ABB RAPID module: StraightAlign3DP.modx

MODULE StraightAlign3DP


	VAR jointtarget CDP_0 := [[-10.64, 35.57, 6.66, 0, 47.77, -100.64], [9E9, 9E9, 9E9, 9E9, 9E9, 9E9]];
	VAR jointtarget CDP_1 := [[-9.53, 35.36, 7.02, 0, 47.62, -99.53], [9E9, 9E9, 9E9, 9E9, 9E9, 9E9]];
	VAR jointtarget CDP_2 := [[-8.41, 35.18, 7.34, 0, 47.48, -98.41], [9E9, 9E9, 9E9, 9E9, 9E9, 9E9]];
	VAR jointtarget CDP_3 := [[-7.29, 35.01, 7.62, 0, 47.37, -97.29], [9E9, 9E9, 9E9, 9E9, 9E9, 9E9]];
	VAR jointtarget CDP_4 := [[-6.16, 34.87, 7.86, 0, 47.27, -96.16], [9E9, 9E9, 9E9, 9E9, 9E9, 9E9]];
	VAR jointtarget CDP_5 := [[-5.02, 34.75, 8.06, 0, 47.19, -95.02], [9E9, 9E9, 9E9, 9E9, 9E9, 9E9]];
	VAR jointtarget CDP_6 := [[-3.89, 34.66, 8.22, 0, 47.12, -93.89], [9E9, 9E9, 9E9, 9E9, 9E9, 9E9]];
	VAR jointtarget CDP_7 := [[-2.75, 34.59, 8.33, 0, 47.07, -92.75], [9E9, 9E9, 9E9, 9E9, 9E9, 9E9]];
	VAR jointtarget CDP_8 := [[-1.6, 34.55, 8.41, 0, 47.04, -91.6], [9E9, 9E9, 9E9, 9E9, 9E9, 9E9]];
	VAR jointtarget CDP_9 := [[-0.46, 34.53, 8.45, 0, 47.03, -90.46], [9E9, 9E9, 9E9, 9E9, 9E9, 9E9]];
	VAR jointtarget CDP_10 := [[0.69, 34.53, 8.44, 0, 47.03, -89.31], [9E9, 9E9, 9E9, 9E9, 9E9, 9E9]];
	VAR jointtarget CDP_11 := [[1.83, 34.55, 8.4, 0, 47.05, -88.17], [9E9, 9E9, 9E9, 9E9, 9E9, 9E9]];
	VAR jointtarget CDP_12 := [[2.97, 34.6, 8.31, 0, 47.08, -87.03], [9E9, 9E9, 9E9, 9E9, 9E9, 9E9]];
	VAR jointtarget CDP_13 := [[4.11, 34.68, 8.19, 0, 47.13, -85.89], [9E9, 9E9, 9E9, 9E9, 9E9, 9E9]];
	VAR jointtarget CDP_14 := [[5.25, 34.78, 8.02, 0, 47.2, -84.75], [9E9, 9E9, 9E9, 9E9, 9E9, 9E9]];
	VAR jointtarget CDP_15 := [[6.38, 34.9, 7.82, 0, 47.29, -83.62], [9E9, 9E9, 9E9, 9E9, 9E9, 9E9]];
	VAR jointtarget CDP_16 := [[7.51, 35.04, 7.57, 0, 47.39, -82.49], [9E9, 9E9, 9E9, 9E9, 9E9, 9E9]];
	VAR jointtarget CDP_17 := [[8.63, 35.21, 7.28, 0, 47.51, -81.37], [9E9, 9E9, 9E9, 9E9, 9E9, 9E9]];
	VAR jointtarget CDP_18 := [[9.75, 35.4, 6.95, 0, 47.64, -80.25], [9E9, 9E9, 9E9, 9E9, 9E9, 9E9]];
	VAR jointtarget CDP_19 := [[10.86, 35.62, 6.58, 0, 47.8, -79.14], [9E9, 9E9, 9E9, 9E9, 9E9, 9E9]];
	VAR jointtarget CDP_20 := [[10.87, 35.62, 6.58, 0, 47.8, -79.46], [9E9, 9E9, 9E9, 9E9, 9E9, 9E9]];
	VAR jointtarget CDP_21 := [[10.89, 35.62, 6.57, 0, 47.8, -80.1], [9E9, 9E9, 9E9, 9E9, 9E9, 9E9]];
	VAR jointtarget CDP_22 := [[10.91, 35.63, 6.57, 0, 47.8, -80.75], [9E9, 9E9, 9E9, 9E9, 9E9, 9E9]];
	VAR jointtarget CDP_23 := [[10.92, 35.63, 6.56, 0, 47.81, -81.39], [9E9, 9E9, 9E9, 9E9, 9E9, 9E9]];
	VAR jointtarget CDP_24 := [[10.94, 35.63, 6.56, 0, 47.81, -82.04], [9E9, 9E9, 9E9, 9E9, 9E9, 9E9]];
	VAR jointtarget CDP_25 := [[10.96, 35.63, 6.56, 0, 47.81, -82.68], [9E9, 9E9, 9E9, 9E9, 9E9, 9E9]];
	VAR jointtarget CDP_26 := [[10.97, 35.64, 6.55, 0, 47.81, -83.33], [9E9, 9E9, 9E9, 9E9, 9E9, 9E9]];
	VAR jointtarget CDP_27 := [[10.99, 35.64, 6.55, 0, 47.81, -83.97], [9E9, 9E9, 9E9, 9E9, 9E9, 9E9]];
	VAR jointtarget CDP_28 := [[11.01, 35.64, 6.55, 0, 47.81, -84.62], [9E9, 9E9, 9E9, 9E9, 9E9, 9E9]];
	VAR jointtarget CDP_29 := [[11.02, 35.64, 6.54, 0, 47.81, -85.27], [9E9, 9E9, 9E9, 9E9, 9E9, 9E9]];
	VAR jointtarget CDP_30 := [[11.04, 35.64, 6.54, 0, 47.82, -85.91], [9E9, 9E9, 9E9, 9E9, 9E9, 9E9]];
	VAR jointtarget CDP_31 := [[11.06, 35.64, 6.54, 0, 47.82, -86.56], [9E9, 9E9, 9E9, 9E9, 9E9, 9E9]];
	VAR jointtarget CDP_32 := [[11.07, 35.65, 6.54, 0, 47.82, -87.2], [9E9, 9E9, 9E9, 9E9, 9E9, 9E9]];
	VAR jointtarget CDP_33 := [[11.09, 35.65, 6.54, 0, 47.82, -87.85], [9E9, 9E9, 9E9, 9E9, 9E9, 9E9]];
	VAR jointtarget CDP_34 := [[11.11, 35.65, 6.54, 0, 47.82, -88.49], [9E9, 9E9, 9E9, 9E9, 9E9, 9E9]];
	VAR jointtarget CDP_35 := [[11.13, 35.65, 6.54, 0, 47.82, -89.14], [9E9, 9E9, 9E9, 9E9, 9E9, 9E9]];
	VAR jointtarget CDP_36 := [[11.14, 35.65, 6.54, 0, 47.82, -89.78], [9E9, 9E9, 9E9, 9E9, 9E9, 9E9]];
	VAR jointtarget CDP_37 := [[11.16, 35.65, 6.54, 0, 47.82, -90.43], [9E9, 9E9, 9E9, 9E9, 9E9, 9E9]];
	VAR jointtarget CDP_38 := [[11.18, 35.65, 6.54, 0, 47.82, -91.07], [9E9, 9E9, 9E9, 9E9, 9E9, 9E9]];
	VAR jointtarget CDP_39 := [[11.19, 35.65, 6.54, 0, 47.82, -91.72], [9E9, 9E9, 9E9, 9E9, 9E9, 9E9]];
	VAR jointtarget CDP_40 := [[11.26, 35.64, 6.54, 0, 47.82, -91.98], [9E9, 9E9, 9E9, 9E9, 9E9, 9E9]];
	VAR jointtarget CDP_41 := [[11.33, 35.64, 6.55, 0, 47.81, -91.91], [9E9, 9E9, 9E9, 9E9, 9E9, 9E9]];
	VAR jointtarget CDP_42 := [[11.4, 35.64, 6.55, 0, 47.81, -91.84], [9E9, 9E9, 9E9, 9E9, 9E9, 9E9]];
	VAR jointtarget CDP_43 := [[11.47, 35.64, 6.55, 0, 47.81, -91.78], [9E9, 9E9, 9E9, 9E9, 9E9, 9E9]];
	VAR jointtarget CDP_44 := [[11.53, 35.63, 6.56, 0, 47.81, -91.71], [9E9, 9E9, 9E9, 9E9, 9E9, 9E9]];
	VAR jointtarget CDP_45 := [[11.6, 35.63, 6.56, 0, 47.81, -91.64], [9E9, 9E9, 9E9, 9E9, 9E9, 9E9]];
	VAR jointtarget CDP_46 := [[11.67, 35.63, 6.56, 0, 47.81, -91.57], [9E9, 9E9, 9E9, 9E9, 9E9, 9E9]];
	VAR jointtarget CDP_47 := [[11.74, 35.63, 6.57, 0, 47.8, -91.5], [9E9, 9E9, 9E9, 9E9, 9E9, 9E9]];
	VAR jointtarget CDP_48 := [[11.81, 35.63, 6.57, 0, 47.8, -91.44], [9E9, 9E9, 9E9, 9E9, 9E9, 9E9]];
	VAR jointtarget CDP_49 := [[11.87, 35.62, 6.57, 0, 47.8, -91.37], [9E9, 9E9, 9E9, 9E9, 9E9, 9E9]];
	VAR jointtarget CDP_50 := [[11.94, 35.62, 6.58, 0, 47.8, -91.3], [9E9, 9E9, 9E9, 9E9, 9E9, 9E9]];
	VAR jointtarget CDP_51 := [[12.01, 35.62, 6.58, 0, 47.8, -91.23], [9E9, 9E9, 9E9, 9E9, 9E9, 9E9]];
	VAR jointtarget CDP_52 := [[12.08, 35.62, 6.58, 0, 47.8, -91.16], [9E9, 9E9, 9E9, 9E9, 9E9, 9E9]];
	VAR jointtarget CDP_53 := [[12.15, 35.62, 6.58, 0, 47.8, -91.09], [9E9, 9E9, 9E9, 9E9, 9E9, 9E9]];
	VAR jointtarget CDP_54 := [[12.21, 35.62, 6.59, 0, 47.8, -91.03], [9E9, 9E9, 9E9, 9E9, 9E9, 9E9]];
	VAR jointtarget CDP_55 := [[12.28, 35.62, 6.59, 0, 47.8, -90.96], [9E9, 9E9, 9E9, 9E9, 9E9, 9E9]];
	VAR jointtarget CDP_56 := [[12.35, 35.61, 6.59, 0, 47.79, -90.89], [9E9, 9E9, 9E9, 9E9, 9E9, 9E9]];
	VAR jointtarget CDP_57 := [[12.42, 35.61, 6.59, 0, 47.79, -90.82], [9E9, 9E9, 9E9, 9E9, 9E9, 9E9]];
	VAR jointtarget CDP_58 := [[12.49, 35.61, 6.59, 0, 47.79, -90.75], [9E9, 9E9, 9E9, 9E9, 9E9, 9E9]];
	VAR jointtarget CDP_59 := [[12.55, 35.61, 6.6, 0, 47.79, -90.69], [9E9, 9E9, 9E9, 9E9, 9E9, 9E9]];
	VAR jointtarget CDP_60 := [[12.69, 35.62, 6.58, 0, 47.8, -85.39], [9E9, 9E9, 9E9, 9E9, 9E9, 9E9]];
	VAR jointtarget CDP_61 := [[12.81, 35.66, 6.51, 0, 47.83, -74.94], [9E9, 9E9, 9E9, 9E9, 9E9, 9E9]];
	VAR jointtarget CDP_62 := [[12.93, 35.72, 6.41, 0, 47.87, -64.5], [9E9, 9E9, 9E9, 9E9, 9E9, 9E9]];
	VAR jointtarget CDP_63 := [[13.04, 35.8, 6.27, 0, 47.93, -54.07], [9E9, 9E9, 9E9, 9E9, 9E9, 9E9]];
	VAR jointtarget CDP_64 := [[13.13, 35.91, 6.09, 0, 48, -43.65], [9E9, 9E9, 9E9, 9E9, 9E9, 9E9]];
	VAR jointtarget CDP_65 := [[13.2, 36.02, 5.89, 0, 48.09, -33.25], [9E9, 9E9, 9E9, 9E9, 9E9, 9E9]];
	VAR jointtarget CDP_66 := [[13.25, 36.16, 5.66, 0, 48.18, -22.88], [9E9, 9E9, 9E9, 9E9, 9E9, 9E9]];
	VAR jointtarget CDP_67 := [[13.28, 36.3, 5.42, 0, 48.28, -12.53], [9E9, 9E9, 9E9, 9E9, 9E9, 9E9]];
	VAR jointtarget CDP_68 := [[13.29, 36.44, 5.18, 0, 48.38, -2.2], [9E9, 9E9, 9E9, 9E9, 9E9, 9E9]];
	VAR jointtarget CDP_69 := [[13.27, 36.58, 4.93, 0, 48.49, 8.11], [9E9, 9E9, 9E9, 9E9, 9E9, 9E9]];
	VAR jointtarget CDP_70 := [[13.23, 36.71, 4.7, 0, 48.58, 18.39], [9E9, 9E9, 9E9, 9E9, 9E9, 9E9]];
	VAR jointtarget CDP_71 := [[13.17, 36.84, 4.48, 0, 48.68, 28.65], [9E9, 9E9, 9E9, 9E9, 9E9, 9E9]];
	VAR jointtarget CDP_72 := [[13.08, 36.95, 4.29, 0, 48.76, 38.9], [9E9, 9E9, 9E9, 9E9, 9E9, 9E9]];
	VAR jointtarget CDP_73 := [[12.99, 37.05, 4.13, 0, 48.82, 49.12], [9E9, 9E9, 9E9, 9E9, 9E9, 9E9]];
	VAR jointtarget CDP_74 := [[12.88, 37.12, 4, 0, 48.88, 59.33], [9E9, 9E9, 9E9, 9E9, 9E9, 9E9]];
	VAR jointtarget CDP_75 := [[12.75, 37.17, 3.92, 0, 48.91, 69.54], [9E9, 9E9, 9E9, 9E9, 9E9, 9E9]];
	VAR jointtarget CDP_76 := [[12.63, 37.19, 3.87, 0, 48.93, 79.73], [9E9, 9E9, 9E9, 9E9, 9E9, 9E9]];
	VAR jointtarget CDP_77 := [[12.5, 37.19, 3.87, 0, 48.93, 89.93], [9E9, 9E9, 9E9, 9E9, 9E9, 9E9]];
	VAR jointtarget CDP_78 := [[12.37, 37.17, 3.92, 0, 48.91, 100.13], [9E9, 9E9, 9E9, 9E9, 9E9, 9E9]];
	VAR jointtarget CDP_79 := [[12.25, 37.12, 4, 0, 48.88, 110.33], [9E9, 9E9, 9E9, 9E9, 9E9, 9E9]];
	VAR jointtarget CDP_80 := [[12.19, 37.09, 4.06, 0, 48.85, 115.43], [9E9, 9E9, 9E9, 9E9, 9E9, 9E9]];
	VAR jointtarget CDP_81 := [[12.13, 37.06, 4.11, 0, 48.83, 115.37], [9E9, 9E9, 9E9, 9E9, 9E9, 9E9]];
	VAR jointtarget CDP_82 := [[12.07, 37.02, 4.17, 0, 48.81, 115.31], [9E9, 9E9, 9E9, 9E9, 9E9, 9E9]];
	VAR jointtarget CDP_83 := [[12.01, 36.99, 4.22, 0, 48.79, 115.25], [9E9, 9E9, 9E9, 9E9, 9E9, 9E9]];
	VAR jointtarget CDP_84 := [[11.95, 36.96, 4.28, 0, 48.76, 115.19], [9E9, 9E9, 9E9, 9E9, 9E9, 9E9]];
	VAR jointtarget CDP_85 := [[11.89, 36.93, 4.33, 0, 48.74, 115.13], [9E9, 9E9, 9E9, 9E9, 9E9, 9E9]];
	VAR jointtarget CDP_86 := [[11.83, 36.9, 4.38, 0, 48.72, 115.07], [9E9, 9E9, 9E9, 9E9, 9E9, 9E9]];
	VAR jointtarget CDP_87 := [[11.77, 36.87, 4.44, 0, 48.7, 115.01], [9E9, 9E9, 9E9, 9E9, 9E9, 9E9]];
	VAR jointtarget CDP_88 := [[11.71, 36.84, 4.49, 0, 48.67, 114.95], [9E9, 9E9, 9E9, 9E9, 9E9, 9E9]];
	VAR jointtarget CDP_89 := [[11.65, 36.81, 4.54, 0, 48.65, 114.89], [9E9, 9E9, 9E9, 9E9, 9E9, 9E9]];
	VAR jointtarget CDP_90 := [[11.59, 36.77, 4.6, 0, 48.63, 114.83], [9E9, 9E9, 9E9, 9E9, 9E9, 9E9]];
	VAR jointtarget CDP_91 := [[11.53, 36.74, 4.65, 0, 48.61, 114.77], [9E9, 9E9, 9E9, 9E9, 9E9, 9E9]];
	VAR jointtarget CDP_92 := [[11.47, 36.71, 4.7, 0, 48.58, 114.71], [9E9, 9E9, 9E9, 9E9, 9E9, 9E9]];
	VAR jointtarget CDP_93 := [[11.4, 36.68, 4.76, 0, 48.56, 114.64], [9E9, 9E9, 9E9, 9E9, 9E9, 9E9]];
	VAR jointtarget CDP_94 := [[11.34, 36.65, 4.81, 0, 48.54, 114.58], [9E9, 9E9, 9E9, 9E9, 9E9, 9E9]];
	VAR jointtarget CDP_95 := [[11.28, 36.62, 4.86, 0, 48.52, 114.52], [9E9, 9E9, 9E9, 9E9, 9E9, 9E9]];
	VAR jointtarget CDP_96 := [[11.22, 36.59, 4.92, 0, 48.49, 114.46], [9E9, 9E9, 9E9, 9E9, 9E9, 9E9]];
	VAR jointtarget CDP_97 := [[11.16, 36.56, 4.97, 0, 48.47, 114.4], [9E9, 9E9, 9E9, 9E9, 9E9, 9E9]];
	VAR jointtarget CDP_98 := [[11.1, 36.53, 5.02, 0, 48.45, 114.34], [9E9, 9E9, 9E9, 9E9, 9E9, 9E9]];
	VAR jointtarget CDP_99 := [[11.04, 36.5, 5.07, 0, 48.43, 114.28], [9E9, 9E9, 9E9, 9E9, 9E9, 9E9]];
	VAR jointtarget CDP_100 := [[11.02, 36.49, 5.08, 0, 48.42, 113.93], [9E9, 9E9, 9E9, 9E9, 9E9, 9E9]];
	VAR jointtarget CDP_101 := [[11.01, 36.48, 5.1, 0, 48.42, 113.26], [9E9, 9E9, 9E9, 9E9, 9E9, 9E9]];
	VAR jointtarget CDP_102 := [[10.99, 36.48, 5.11, 0, 48.41, 112.58], [9E9, 9E9, 9E9, 9E9, 9E9, 9E9]];
	VAR jointtarget CDP_103 := [[10.98, 36.47, 5.12, 0, 48.41, 111.9], [9E9, 9E9, 9E9, 9E9, 9E9, 9E9]];
	VAR jointtarget CDP_104 := [[10.96, 36.46, 5.13, 0, 48.4, 111.22], [9E9, 9E9, 9E9, 9E9, 9E9, 9E9]];
	VAR jointtarget CDP_105 := [[10.95, 36.46, 5.14, 0, 48.4, 110.55], [9E9, 9E9, 9E9, 9E9, 9E9, 9E9]];
	VAR jointtarget CDP_106 := [[10.93, 36.45, 5.15, 0, 48.39, 109.87], [9E9, 9E9, 9E9, 9E9, 9E9, 9E9]];
	VAR jointtarget CDP_107 := [[10.91, 36.45, 5.16, 0, 48.39, 109.19], [9E9, 9E9, 9E9, 9E9, 9E9, 9E9]];
	VAR jointtarget CDP_108 := [[10.9, 36.44, 5.17, 0, 48.39, 108.51], [9E9, 9E9, 9E9, 9E9, 9E9, 9E9]];
	VAR jointtarget CDP_109 := [[10.88, 36.43, 5.18, 0, 48.38, 107.83], [9E9, 9E9, 9E9, 9E9, 9E9, 9E9]];
	VAR jointtarget CDP_110 := [[10.87, 36.43, 5.19, 0, 48.38, 107.16], [9E9, 9E9, 9E9, 9E9, 9E9, 9E9]];
	VAR jointtarget CDP_111 := [[10.85, 36.42, 5.2, 0, 48.37, 106.48], [9E9, 9E9, 9E9, 9E9, 9E9, 9E9]];
	VAR jointtarget CDP_112 := [[10.83, 36.42, 5.21, 0, 48.37, 105.8], [9E9, 9E9, 9E9, 9E9, 9E9, 9E9]];
	VAR jointtarget CDP_113 := [[10.82, 36.41, 5.22, 0, 48.37, 105.12], [9E9, 9E9, 9E9, 9E9, 9E9, 9E9]];
	VAR jointtarget CDP_114 := [[10.8, 36.41, 5.23, 0, 48.36, 104.44], [9E9, 9E9, 9E9, 9E9, 9E9, 9E9]];
	VAR jointtarget CDP_115 := [[10.79, 36.4, 5.23, 0, 48.36, 103.77], [9E9, 9E9, 9E9, 9E9, 9E9, 9E9]];
	VAR jointtarget CDP_116 := [[10.77, 36.4, 5.24, 0, 48.36, 103.09], [9E9, 9E9, 9E9, 9E9, 9E9, 9E9]];
	VAR jointtarget CDP_117 := [[10.75, 36.4, 5.25, 0, 48.36, 102.41], [9E9, 9E9, 9E9, 9E9, 9E9, 9E9]];
	VAR jointtarget CDP_118 := [[10.74, 36.39, 5.25, 0, 48.35, 101.73], [9E9, 9E9, 9E9, 9E9, 9E9, 9E9]];
	VAR jointtarget CDP_119 := [[10.72, 36.39, 5.26, 0, 48.35, 101.05], [9E9, 9E9, 9E9, 9E9, 9E9, 9E9]];
	VAR jointtarget CDP_120 := [[9.64, 36.18, 5.62, 0, 48.2, 99.64], [9E9, 9E9, 9E9, 9E9, 9E9, 9E9]];
	VAR jointtarget CDP_121 := [[8.56, 35.99, 5.95, 0, 48.06, 98.56], [9E9, 9E9, 9E9, 9E9, 9E9, 9E9]];
	VAR jointtarget CDP_122 := [[7.47, 35.83, 6.23, 0, 47.95, 97.47], [9E9, 9E9, 9E9, 9E9, 9E9, 9E9]];
	VAR jointtarget CDP_123 := [[6.38, 35.68, 6.47, 0, 47.84, 96.38], [9E9, 9E9, 9E9, 9E9, 9E9, 9E9]];
	VAR jointtarget CDP_124 := [[5.28, 35.56, 6.68, 0, 47.76, 95.28], [9E9, 9E9, 9E9, 9E9, 9E9, 9E9]];
	VAR jointtarget CDP_125 := [[4.17, 35.46, 6.85, 0, 47.69, 94.17], [9E9, 9E9, 9E9, 9E9, 9E9, 9E9]];
	VAR jointtarget CDP_126 := [[3.07, 35.39, 6.97, 0, 47.64, 93.07], [9E9, 9E9, 9E9, 9E9, 9E9, 9E9]];
	VAR jointtarget CDP_127 := [[1.96, 35.34, 7.06, 0, 47.6, 91.96], [9E9, 9E9, 9E9, 9E9, 9E9, 9E9]];
	VAR jointtarget CDP_128 := [[0.85, 35.31, 7.11, 0, 47.58, 90.85], [9E9, 9E9, 9E9, 9E9, 9E9, 9E9]];
	VAR jointtarget CDP_129 := [[-0.26, 35.3, 7.12, 0, 47.57, 89.74], [9E9, 9E9, 9E9, 9E9, 9E9, 9E9]];
	VAR jointtarget CDP_130 := [[-1.37, 35.32, 7.09, 0, 47.59, 88.63], [9E9, 9E9, 9E9, 9E9, 9E9, 9E9]];
	VAR jointtarget CDP_131 := [[-2.48, 35.36, 7.03, 0, 47.61, 87.52], [9E9, 9E9, 9E9, 9E9, 9E9, 9E9]];
	VAR jointtarget CDP_132 := [[-3.59, 35.42, 6.92, 0, 47.66, 86.41], [9E9, 9E9, 9E9, 9E9, 9E9, 9E9]];
	VAR jointtarget CDP_133 := [[-4.7, 35.51, 6.77, 0, 47.72, 85.3], [9E9, 9E9, 9E9, 9E9, 9E9, 9E9]];
	VAR jointtarget CDP_134 := [[-5.8, 35.62, 6.59, 0, 47.8, 84.2], [9E9, 9E9, 9E9, 9E9, 9E9, 9E9]];
	VAR jointtarget CDP_135 := [[-6.9, 35.75, 6.36, 0, 47.89, 83.1], [9E9, 9E9, 9E9, 9E9, 9E9, 9E9]];
	VAR jointtarget CDP_136 := [[-7.99, 35.9, 6.1, 0, 48, 82.01], [9E9, 9E9, 9E9, 9E9, 9E9, 9E9]];
	VAR jointtarget CDP_137 := [[-9.08, 36.08, 5.8, 0, 48.13, 80.92], [9E9, 9E9, 9E9, 9E9, 9E9, 9E9]];
	VAR jointtarget CDP_138 := [[-10.16, 36.28, 5.46, 0, 48.27, 79.84], [9E9, 9E9, 9E9, 9E9, 9E9, 9E9]];
	VAR jointtarget CDP_139 := [[-11.23, 36.5, 5.07, 0, 48.43, 78.77], [9E9, 9E9, 9E9, 9E9, 9E9, 9E9]];
	VAR jointtarget CDP_140 := [[-11.28, 36.51, 5.06, 0, 48.44, 79.81], [9E9, 9E9, 9E9, 9E9, 9E9, 9E9]];
	VAR jointtarget CDP_141 := [[-11.34, 36.52, 5.04, 0, 48.44, 81.95], [9E9, 9E9, 9E9, 9E9, 9E9, 9E9]];
	VAR jointtarget CDP_142 := [[-11.39, 36.52, 5.03, 0, 48.45, 84.09], [9E9, 9E9, 9E9, 9E9, 9E9, 9E9]];
	VAR jointtarget CDP_143 := [[-11.45, 36.53, 5.02, 0, 48.45, 86.23], [9E9, 9E9, 9E9, 9E9, 9E9, 9E9]];
	VAR jointtarget CDP_144 := [[-11.5, 36.53, 5.02, 0, 48.45, 88.37], [9E9, 9E9, 9E9, 9E9, 9E9, 9E9]];
	VAR jointtarget CDP_145 := [[-11.56, 36.53, 5.02, 0, 48.45, 90.51], [9E9, 9E9, 9E9, 9E9, 9E9, 9E9]];
	VAR jointtarget CDP_146 := [[-11.61, 36.53, 5.03, 0, 48.45, 92.65], [9E9, 9E9, 9E9, 9E9, 9E9, 9E9]];
	VAR jointtarget CDP_147 := [[-11.67, 36.52, 5.04, 0, 48.44, 94.78], [9E9, 9E9, 9E9, 9E9, 9E9, 9E9]];
	VAR jointtarget CDP_148 := [[-11.72, 36.51, 5.05, 0, 48.44, 96.92], [9E9, 9E9, 9E9, 9E9, 9E9, 9E9]];
	VAR jointtarget CDP_149 := [[-11.78, 36.5, 5.06, 0, 48.43, 99.06], [9E9, 9E9, 9E9, 9E9, 9E9, 9E9]];
	VAR jointtarget CDP_150 := [[-11.83, 36.49, 5.09, 0, 48.42, 101.2], [9E9, 9E9, 9E9, 9E9, 9E9, 9E9]];
	VAR jointtarget CDP_151 := [[-11.89, 36.48, 5.11, 0, 48.41, 103.34], [9E9, 9E9, 9E9, 9E9, 9E9, 9E9]];
	VAR jointtarget CDP_152 := [[-11.94, 36.46, 5.14, 0, 48.4, 105.48], [9E9, 9E9, 9E9, 9E9, 9E9, 9E9]];
	VAR jointtarget CDP_153 := [[-11.99, 36.44, 5.17, 0, 48.39, 107.63], [9E9, 9E9, 9E9, 9E9, 9E9, 9E9]];
	VAR jointtarget CDP_154 := [[-12.04, 36.42, 5.2, 0, 48.37, 109.77], [9E9, 9E9, 9E9, 9E9, 9E9, 9E9]];
	VAR jointtarget CDP_155 := [[-12.09, 36.4, 5.24, 0, 48.36, 111.91], [9E9, 9E9, 9E9, 9E9, 9E9, 9E9]];
	VAR jointtarget CDP_156 := [[-12.15, 36.38, 5.28, 0, 48.34, 114.05], [9E9, 9E9, 9E9, 9E9, 9E9, 9E9]];
	VAR jointtarget CDP_157 := [[-12.19, 36.35, 5.33, 0, 48.32, 116.2], [9E9, 9E9, 9E9, 9E9, 9E9, 9E9]];
	VAR jointtarget CDP_158 := [[-12.24, 36.32, 5.38, 0, 48.3, 118.34], [9E9, 9E9, 9E9, 9E9, 9E9, 9E9]];
	VAR jointtarget CDP_159 := [[-12.29, 36.29, 5.43, 0, 48.28, 120.49], [9E9, 9E9, 9E9, 9E9, 9E9, 9E9]];
	VAR jointtarget CDP_160 := [[-12.32, 36.27, 5.47, 0, 48.26, 121.56], [9E9, 9E9, 9E9, 9E9, 9E9, 9E9]];
	VAR jointtarget CDP_161 := [[-12.35, 36.25, 5.5, 0, 48.25, 121.53], [9E9, 9E9, 9E9, 9E9, 9E9, 9E9]];
	VAR jointtarget CDP_162 := [[-12.38, 36.23, 5.53, 0, 48.24, 121.5], [9E9, 9E9, 9E9, 9E9, 9E9, 9E9]];
	VAR jointtarget CDP_163 := [[-12.41, 36.21, 5.56, 0, 48.22, 121.47], [9E9, 9E9, 9E9, 9E9, 9E9, 9E9]];
	VAR jointtarget CDP_164 := [[-12.43, 36.19, 5.6, 0, 48.21, 121.44], [9E9, 9E9, 9E9, 9E9, 9E9, 9E9]];
	VAR jointtarget CDP_165 := [[-12.46, 36.18, 5.63, 0, 48.2, 121.41], [9E9, 9E9, 9E9, 9E9, 9E9, 9E9]];
	VAR jointtarget CDP_166 := [[-12.49, 36.16, 5.66, 0, 48.18, 121.39], [9E9, 9E9, 9E9, 9E9, 9E9, 9E9]];
	VAR jointtarget CDP_167 := [[-12.52, 36.14, 5.69, 0, 48.17, 121.36], [9E9, 9E9, 9E9, 9E9, 9E9, 9E9]];
	VAR jointtarget CDP_168 := [[-12.55, 36.12, 5.73, 0, 48.16, 121.33], [9E9, 9E9, 9E9, 9E9, 9E9, 9E9]];
	VAR jointtarget CDP_169 := [[-12.58, 36.1, 5.76, 0, 48.14, 121.3], [9E9, 9E9, 9E9, 9E9, 9E9, 9E9]];
	VAR jointtarget CDP_170 := [[-12.61, 36.08, 5.79, 0, 48.13, 121.27], [9E9, 9E9, 9E9, 9E9, 9E9, 9E9]];
	VAR jointtarget CDP_171 := [[-12.63, 36.06, 5.82, 0, 48.11, 121.24], [9E9, 9E9, 9E9, 9E9, 9E9, 9E9]];
	VAR jointtarget CDP_172 := [[-12.66, 36.04, 5.86, 0, 48.1, 121.21], [9E9, 9E9, 9E9, 9E9, 9E9, 9E9]];
	VAR jointtarget CDP_173 := [[-12.69, 36.02, 5.89, 0, 48.09, 121.18], [9E9, 9E9, 9E9, 9E9, 9E9, 9E9]];
	VAR jointtarget CDP_174 := [[-12.72, 36.01, 5.92, 0, 48.07, 121.16], [9E9, 9E9, 9E9, 9E9, 9E9, 9E9]];
	VAR jointtarget CDP_175 := [[-12.75, 35.99, 5.95, 0, 48.06, 121.13], [9E9, 9E9, 9E9, 9E9, 9E9, 9E9]];
	VAR jointtarget CDP_176 := [[-12.78, 35.97, 5.99, 0, 48.05, 121.1], [9E9, 9E9, 9E9, 9E9, 9E9, 9E9]];
	VAR jointtarget CDP_177 := [[-12.81, 35.95, 6.02, 0, 48.03, 121.07], [9E9, 9E9, 9E9, 9E9, 9E9, 9E9]];
	VAR jointtarget CDP_178 := [[-12.84, 35.93, 6.05, 0, 48.02, 121.04], [9E9, 9E9, 9E9, 9E9, 9E9, 9E9]];
	VAR jointtarget CDP_179 := [[-12.86, 35.91, 6.08, 0, 48.01, 121.01], [9E9, 9E9, 9E9, 9E9, 9E9, 9E9]];
	VAR jointtarget CDP_180 := [[-13.02, 35.84, 6.21, 0, 47.95, 114.17], [9E9, 9E9, 9E9, 9E9, 9E9, 9E9]];
	VAR jointtarget CDP_181 := [[-13.18, 35.81, 6.26, 0, 47.93, 100.62], [9E9, 9E9, 9E9, 9E9, 9E9, 9E9]];
	VAR jointtarget CDP_182 := [[-13.34, 35.81, 6.25, 0, 47.94, 87.07], [9E9, 9E9, 9E9, 9E9, 9E9, 9E9]];
	VAR jointtarget CDP_183 := [[-13.5, 35.86, 6.16, 0, 47.97, 73.52], [9E9, 9E9, 9E9, 9E9, 9E9, 9E9]];
	VAR jointtarget CDP_184 := [[-13.64, 35.95, 6.01, 0, 48.04, 59.99], [9E9, 9E9, 9E9, 9E9, 9E9, 9E9]];
	VAR jointtarget CDP_185 := [[-13.76, 36.08, 5.8, 0, 48.12, 46.48], [9E9, 9E9, 9E9, 9E9, 9E9, 9E9]];
	VAR jointtarget CDP_186 := [[-13.85, 36.22, 5.54, 0, 48.23, 33.01], [9E9, 9E9, 9E9, 9E9, 9E9, 9E9]];
	VAR jointtarget CDP_187 := [[-13.91, 36.39, 5.26, 0, 48.35, 19.56], [9E9, 9E9, 9E9, 9E9, 9E9, 9E9]];
	VAR jointtarget CDP_188 := [[-13.92, 36.57, 4.95, 0, 48.48, 6.16], [9E9, 9E9, 9E9, 9E9, 9E9, 9E9]];
	VAR jointtarget CDP_189 := [[-13.9, 36.75, 4.64, 0, 48.61, -7.21], [9E9, 9E9, 9E9, 9E9, 9E9, 9E9]];
	VAR jointtarget CDP_190 := [[-13.85, 36.92, 4.36, 0, 48.73, -20.54], [9E9, 9E9, 9E9, 9E9, 9E9, 9E9]];
	VAR jointtarget CDP_191 := [[-13.76, 37.06, 4.1, 0, 48.84, -33.84], [9E9, 9E9, 9E9, 9E9, 9E9, 9E9]];
	VAR jointtarget CDP_192 := [[-13.64, 37.19, 3.89, 0, 48.93, -47.11], [9E9, 9E9, 9E9, 9E9, 9E9, 9E9]];
	VAR jointtarget CDP_193 := [[-13.5, 37.27, 3.73, 0, 48.99, -60.35], [9E9, 9E9, 9E9, 9E9, 9E9, 9E9]];
	VAR jointtarget CDP_194 := [[-13.34, 37.33, 3.65, 0, 49.03, -73.59], [9E9, 9E9, 9E9, 9E9, 9E9, 9E9]];
	VAR jointtarget CDP_195 := [[-13.18, 37.34, 3.63, 0, 49.04, -86.81], [9E9, 9E9, 9E9, 9E9, 9E9, 9E9]];
	VAR jointtarget CDP_196 := [[-13.02, 37.3, 3.68, 0, 49.01, -100.04], [9E9, 9E9, 9E9, 9E9, 9E9, 9E9]];
	VAR jointtarget CDP_197 := [[-12.88, 37.23, 3.81, 0, 48.96, -113.28], [9E9, 9E9, 9E9, 9E9, 9E9, 9E9]];
	VAR jointtarget CDP_198 := [[-12.75, 37.13, 3.99, 0, 48.88, -126.54], [9E9, 9E9, 9E9, 9E9, 9E9, 9E9]];
	VAR jointtarget CDP_199 := [[-12.64, 36.99, 4.23, 0, 48.78, -139.82], [9E9, 9E9, 9E9, 9E9, 9E9, 9E9]];
	VAR jointtarget CDP_200 := [[-12.62, 36.95, 4.3, 0, 48.75, -146.49], [9E9, 9E9, 9E9, 9E9, 9E9, 9E9]];
	VAR jointtarget CDP_201 := [[-12.59, 36.91, 4.37, 0, 48.72, -146.47], [9E9, 9E9, 9E9, 9E9, 9E9, 9E9]];
	VAR jointtarget CDP_202 := [[-12.57, 36.86, 4.44, 0, 48.69, -146.44], [9E9, 9E9, 9E9, 9E9, 9E9, 9E9]];
	VAR jointtarget CDP_203 := [[-12.54, 36.82, 4.51, 0, 48.66, -146.42], [9E9, 9E9, 9E9, 9E9, 9E9, 9E9]];
	VAR jointtarget CDP_204 := [[-12.52, 36.78, 4.58, 0, 48.63, -146.4], [9E9, 9E9, 9E9, 9E9, 9E9, 9E9]];
	VAR jointtarget CDP_205 := [[-12.49, 36.74, 4.65, 0, 48.6, -146.37], [9E9, 9E9, 9E9, 9E9, 9E9, 9E9]];
	VAR jointtarget CDP_206 := [[-12.47, 36.7, 4.73, 0, 48.57, -146.35], [9E9, 9E9, 9E9, 9E9, 9E9, 9E9]];
	VAR jointtarget CDP_207 := [[-12.44, 36.66, 4.8, 0, 48.54, -146.32], [9E9, 9E9, 9E9, 9E9, 9E9, 9E9]];
	VAR jointtarget CDP_208 := [[-12.42, 36.62, 4.87, 0, 48.52, -146.3], [9E9, 9E9, 9E9, 9E9, 9E9, 9E9]];
	VAR jointtarget CDP_209 := [[-12.39, 36.58, 4.94, 0, 48.49, -146.27], [9E9, 9E9, 9E9, 9E9, 9E9, 9E9]];
	VAR jointtarget CDP_210 := [[-12.37, 36.54, 5.01, 0, 48.46, -146.25], [9E9, 9E9, 9E9, 9E9, 9E9, 9E9]];
	VAR jointtarget CDP_211 := [[-12.34, 36.5, 5.08, 0, 48.43, -146.22], [9E9, 9E9, 9E9, 9E9, 9E9, 9E9]];
	VAR jointtarget CDP_212 := [[-12.32, 36.45, 5.15, 0, 48.4, -146.2], [9E9, 9E9, 9E9, 9E9, 9E9, 9E9]];
	VAR jointtarget CDP_213 := [[-12.29, 36.41, 5.22, 0, 48.37, -146.17], [9E9, 9E9, 9E9, 9E9, 9E9, 9E9]];
	VAR jointtarget CDP_214 := [[-12.27, 36.37, 5.29, 0, 48.34, -146.15], [9E9, 9E9, 9E9, 9E9, 9E9, 9E9]];
	VAR jointtarget CDP_215 := [[-12.24, 36.33, 5.36, 0, 48.31, -146.12], [9E9, 9E9, 9E9, 9E9, 9E9, 9E9]];
	VAR jointtarget CDP_216 := [[-12.22, 36.29, 5.43, 0, 48.28, -146.1], [9E9, 9E9, 9E9, 9E9, 9E9, 9E9]];
	VAR jointtarget CDP_217 := [[-12.19, 36.25, 5.5, 0, 48.25, -146.07], [9E9, 9E9, 9E9, 9E9, 9E9, 9E9]];
	VAR jointtarget CDP_218 := [[-12.17, 36.21, 5.57, 0, 48.22, -146.05], [9E9, 9E9, 9E9, 9E9, 9E9, 9E9]];
	VAR jointtarget CDP_219 := [[-12.14, 36.17, 5.64, 0, 48.19, -146.02], [9E9, 9E9, 9E9, 9E9, 9E9, 9E9]];
	VAR jointtarget CDP_220 := [[-12.14, 36.16, 5.66, 0, 48.18, -145.46], [9E9, 9E9, 9E9, 9E9, 9E9, 9E9]];
	VAR jointtarget CDP_221 := [[-12.13, 36.14, 5.68, 0, 48.17, -144.35], [9E9, 9E9, 9E9, 9E9, 9E9, 9E9]];
	VAR jointtarget CDP_222 := [[-12.12, 36.13, 5.7, 0, 48.17, -143.24], [9E9, 9E9, 9E9, 9E9, 9E9, 9E9]];
	VAR jointtarget CDP_223 := [[-12.11, 36.12, 5.72, 0, 48.16, -142.13], [9E9, 9E9, 9E9, 9E9, 9E9, 9E9]];
	VAR jointtarget CDP_224 := [[-12.1, 36.11, 5.74, 0, 48.15, -141.01], [9E9, 9E9, 9E9, 9E9, 9E9, 9E9]];
	VAR jointtarget CDP_225 := [[-12.09, 36.1, 5.76, 0, 48.14, -139.9], [9E9, 9E9, 9E9, 9E9, 9E9, 9E9]];
	VAR jointtarget CDP_226 := [[-12.08, 36.08, 5.78, 0, 48.13, -138.79], [9E9, 9E9, 9E9, 9E9, 9E9, 9E9]];
	VAR jointtarget CDP_227 := [[-12.07, 36.07, 5.8, 0, 48.12, -137.68], [9E9, 9E9, 9E9, 9E9, 9E9, 9E9]];
	VAR jointtarget CDP_228 := [[-12.06, 36.06, 5.82, 0, 48.12, -136.56], [9E9, 9E9, 9E9, 9E9, 9E9, 9E9]];
	VAR jointtarget CDP_229 := [[-12.05, 36.05, 5.84, 0, 48.11, -135.45], [9E9, 9E9, 9E9, 9E9, 9E9, 9E9]];
	VAR jointtarget CDP_230 := [[-12.04, 36.04, 5.86, 0, 48.1, -134.34], [9E9, 9E9, 9E9, 9E9, 9E9, 9E9]];
	VAR jointtarget CDP_231 := [[-12.03, 36.03, 5.88, 0, 48.09, -133.22], [9E9, 9E9, 9E9, 9E9, 9E9, 9E9]];
	VAR jointtarget CDP_232 := [[-12.02, 36.02, 5.89, 0, 48.09, -132.11], [9E9, 9E9, 9E9, 9E9, 9E9, 9E9]];
	VAR jointtarget CDP_233 := [[-12.01, 36.01, 5.91, 0, 48.08, -130.99], [9E9, 9E9, 9E9, 9E9, 9E9, 9E9]];
	VAR jointtarget CDP_234 := [[-12, 36, 5.93, 0, 48.07, -129.88], [9E9, 9E9, 9E9, 9E9, 9E9, 9E9]];
	VAR jointtarget CDP_235 := [[-11.99, 35.99, 5.94, 0, 48.07, -128.76], [9E9, 9E9, 9E9, 9E9, 9E9, 9E9]];
	VAR jointtarget CDP_236 := [[-11.98, 35.98, 5.96, 0, 48.06, -127.65], [9E9, 9E9, 9E9, 9E9, 9E9, 9E9]];
	VAR jointtarget CDP_237 := [[-11.97, 35.97, 5.97, 0, 48.06, -126.53], [9E9, 9E9, 9E9, 9E9, 9E9, 9E9]];
	VAR jointtarget CDP_238 := [[-11.96, 35.96, 5.99, 0, 48.05, -125.42], [9E9, 9E9, 9E9, 9E9, 9E9, 9E9]];
	VAR jointtarget CDP_239 := [[-11.95, 35.95, 6, 0, 48.04, -124.3], [9E9, 9E9, 9E9, 9E9, 9E9, 9E9]];
	VAR jointtarget CDP_240 := [[-11.94, 35.94, 6.02, 0, 48.04, -123.74], [9E9, 9E9, 9E9, 9E9, 9E9, 9E9]];
	VAR jointtarget CDP_241 := [[-11.93, 35.94, 6.03, 0, 48.04, -123.73], [9E9, 9E9, 9E9, 9E9, 9E9, 9E9]];
	VAR jointtarget CDP_242 := [[-11.92, 35.93, 6.04, 0, 48.03, -123.72], [9E9, 9E9, 9E9, 9E9, 9E9, 9E9]];
	VAR jointtarget CDP_243 := [[-11.9, 35.92, 6.05, 0, 48.03, -123.71], [9E9, 9E9, 9E9, 9E9, 9E9, 9E9]];
	VAR jointtarget CDP_244 := [[-11.89, 35.91, 6.07, 0, 48.02, -123.7], [9E9, 9E9, 9E9, 9E9, 9E9, 9E9]];
	VAR jointtarget CDP_245 := [[-11.88, 35.9, 6.08, 0, 48.02, -123.69], [9E9, 9E9, 9E9, 9E9, 9E9, 9E9]];
	VAR jointtarget CDP_246 := [[-11.87, 35.9, 6.09, 0, 48.01, -123.68], [9E9, 9E9, 9E9, 9E9, 9E9, 9E9]];
	VAR jointtarget CDP_247 := [[-11.86, 35.89, 6.11, 0, 48.01, -123.66], [9E9, 9E9, 9E9, 9E9, 9E9, 9E9]];
	VAR jointtarget CDP_248 := [[-11.85, 35.88, 6.12, 0, 48, -123.65], [9E9, 9E9, 9E9, 9E9, 9E9, 9E9]];
	VAR jointtarget CDP_249 := [[-11.84, 35.87, 6.13, 0, 48, -123.64], [9E9, 9E9, 9E9, 9E9, 9E9, 9E9]];
	VAR jointtarget CDP_250 := [[-11.83, 35.86, 6.14, 0, 47.99, -123.63], [9E9, 9E9, 9E9, 9E9, 9E9, 9E9]];
	VAR jointtarget CDP_251 := [[-11.82, 35.86, 6.16, 0, 47.99, -123.62], [9E9, 9E9, 9E9, 9E9, 9E9, 9E9]];
	VAR jointtarget CDP_252 := [[-11.81, 35.85, 6.17, 0, 47.98, -123.61], [9E9, 9E9, 9E9, 9E9, 9E9, 9E9]];
	VAR jointtarget CDP_253 := [[-11.8, 35.84, 6.18, 0, 47.98, -123.6], [9E9, 9E9, 9E9, 9E9, 9E9, 9E9]];
	VAR jointtarget CDP_254 := [[-11.79, 35.83, 6.19, 0, 47.97, -123.59], [9E9, 9E9, 9E9, 9E9, 9E9, 9E9]];
	VAR jointtarget CDP_255 := [[-11.78, 35.83, 6.21, 0, 47.97, -123.58], [9E9, 9E9, 9E9, 9E9, 9E9, 9E9]];
	VAR jointtarget CDP_256 := [[-11.77, 35.82, 6.22, 0, 47.96, -123.57], [9E9, 9E9, 9E9, 9E9, 9E9, 9E9]];
	VAR jointtarget CDP_257 := [[-11.76, 35.81, 6.23, 0, 47.96, -123.56], [9E9, 9E9, 9E9, 9E9, 9E9, 9E9]];
	VAR jointtarget CDP_258 := [[-11.75, 35.8, 6.25, 0, 47.95, -123.55], [9E9, 9E9, 9E9, 9E9, 9E9, 9E9]];
	VAR jointtarget CDP_259 := [[-11.74, 35.79, 6.26, 0, 47.95, -123.54], [9E9, 9E9, 9E9, 9E9, 9E9, 9E9]];
	VAR jointtarget CDP_260 := [[-10.65, 35.56, 6.66, 0, 47.78, -100.65], [9E9, 9E9, 9E9, 9E9, 9E9, 9E9]];
	VAR jointtarget CDP_261 := [[-9.55, 35.35, 7.01, 0, 47.63, -99.55], [9E9, 9E9, 9E9, 9E9, 9E9, 9E9]];
	VAR jointtarget CDP_262 := [[-8.44, 35.17, 7.33, 0, 47.5, -98.44], [9E9, 9E9, 9E9, 9E9, 9E9, 9E9]];
	VAR jointtarget CDP_263 := [[-7.33, 35, 7.61, 0, 47.39, -97.33], [9E9, 9E9, 9E9, 9E9, 9E9, 9E9]];
	VAR jointtarget CDP_264 := [[-6.21, 34.86, 7.85, 0, 47.29, -96.21], [9E9, 9E9, 9E9, 9E9, 9E9, 9E9]];
	VAR jointtarget CDP_265 := [[-5.09, 34.75, 8.05, 0, 47.21, -95.09], [9E9, 9E9, 9E9, 9E9, 9E9, 9E9]];
	VAR jointtarget CDP_266 := [[-3.96, 34.65, 8.21, 0, 47.14, -93.96], [9E9, 9E9, 9E9, 9E9, 9E9, 9E9]];
	VAR jointtarget CDP_267 := [[-2.83, 34.58, 8.33, 0, 47.09, -92.83], [9E9, 9E9, 9E9, 9E9, 9E9, 9E9]];
	VAR jointtarget CDP_268 := [[-1.7, 34.54, 8.4, 0, 47.06, -91.7], [9E9, 9E9, 9E9, 9E9, 9E9, 9E9]];
	VAR jointtarget CDP_269 := [[-0.56, 34.51, 8.44, 0, 47.04, -90.56], [9E9, 9E9, 9E9, 9E9, 9E9, 9E9]];
	VAR jointtarget CDP_270 := [[0.57, 34.51, 8.44, 0, 47.04, -89.43], [9E9, 9E9, 9E9, 9E9, 9E9, 9E9]];
	VAR jointtarget CDP_271 := [[1.7, 34.54, 8.4, 0, 47.06, -88.3], [9E9, 9E9, 9E9, 9E9, 9E9, 9E9]];
	VAR jointtarget CDP_272 := [[2.84, 34.58, 8.32, 0, 47.09, -87.16], [9E9, 9E9, 9E9, 9E9, 9E9, 9E9]];
	VAR jointtarget CDP_273 := [[3.97, 34.65, 8.2, 0, 47.14, -86.03], [9E9, 9E9, 9E9, 9E9, 9E9, 9E9]];
	VAR jointtarget CDP_274 := [[5.09, 34.75, 8.05, 0, 47.21, -84.91], [9E9, 9E9, 9E9, 9E9, 9E9, 9E9]];
	VAR jointtarget CDP_275 := [[6.22, 34.86, 7.85, 0, 47.29, -83.78], [9E9, 9E9, 9E9, 9E9, 9E9, 9E9]];
	VAR jointtarget CDP_276 := [[7.34, 35, 7.61, 0, 47.39, -82.66], [9E9, 9E9, 9E9, 9E9, 9E9, 9E9]];
	VAR jointtarget CDP_277 := [[8.45, 35.17, 7.33, 0, 47.5, -81.55], [9E9, 9E9, 9E9, 9E9, 9E9, 9E9]];
	VAR jointtarget CDP_278 := [[9.56, 35.35, 7.01, 0, 47.64, -80.44], [9E9, 9E9, 9E9, 9E9, 9E9, 9E9]];
	VAR jointtarget CDP_279 := [[10.65, 35.56, 6.65, 0, 47.78, -79.35], [9E9, 9E9, 9E9, 9E9, 9E9, 9E9]];
	VAR jointtarget CDP_280 := [[10.71, 35.58, 6.63, 0, 47.79, -78.19], [9E9, 9E9, 9E9, 9E9, 9E9, 9E9]];
	VAR jointtarget CDP_281 := [[10.76, 35.59, 6.61, 0, 47.8, -75.95], [9E9, 9E9, 9E9, 9E9, 9E9, 9E9]];
	VAR jointtarget CDP_282 := [[10.82, 35.61, 6.58, 0, 47.82, -73.7], [9E9, 9E9, 9E9, 9E9, 9E9, 9E9]];
	VAR jointtarget CDP_283 := [[10.87, 35.63, 6.55, 0, 47.83, -71.45], [9E9, 9E9, 9E9, 9E9, 9E9, 9E9]];
	VAR jointtarget CDP_284 := [[10.92, 35.65, 6.51, 0, 47.84, -69.2], [9E9, 9E9, 9E9, 9E9, 9E9, 9E9]];
	VAR jointtarget CDP_285 := [[10.97, 35.67, 6.47, 0, 47.86, -66.96], [9E9, 9E9, 9E9, 9E9, 9E9, 9E9]];
	VAR jointtarget CDP_286 := [[11.03, 35.7, 6.42, 0, 47.88, -64.72], [9E9, 9E9, 9E9, 9E9, 9E9, 9E9]];
	VAR jointtarget CDP_287 := [[11.07, 35.72, 6.38, 0, 47.9, -62.47], [9E9, 9E9, 9E9, 9E9, 9E9, 9E9]];
	VAR jointtarget CDP_288 := [[11.12, 35.75, 6.33, 0, 47.92, -60.23], [9E9, 9E9, 9E9, 9E9, 9E9, 9E9]];
	VAR jointtarget CDP_289 := [[11.17, 35.79, 6.27, 0, 47.94, -57.99], [9E9, 9E9, 9E9, 9E9, 9E9, 9E9]];
	VAR jointtarget CDP_290 := [[11.22, 35.82, 6.21, 0, 47.97, -55.75], [9E9, 9E9, 9E9, 9E9, 9E9, 9E9]];
	VAR jointtarget CDP_291 := [[11.26, 35.86, 6.15, 0, 47.99, -53.51], [9E9, 9E9, 9E9, 9E9, 9E9, 9E9]];
	VAR jointtarget CDP_292 := [[11.3, 35.89, 6.09, 0, 48.02, -51.27], [9E9, 9E9, 9E9, 9E9, 9E9, 9E9]];
	VAR jointtarget CDP_293 := [[11.35, 35.93, 6.02, 0, 48.05, -49.04], [9E9, 9E9, 9E9, 9E9, 9E9, 9E9]];
	VAR jointtarget CDP_294 := [[11.39, 35.97, 5.95, 0, 48.08, -46.8], [9E9, 9E9, 9E9, 9E9, 9E9, 9E9]];
	VAR jointtarget CDP_295 := [[11.43, 36.02, 5.88, 0, 48.11, -44.57], [9E9, 9E9, 9E9, 9E9, 9E9, 9E9]];
	VAR jointtarget CDP_296 := [[11.46, 36.06, 5.8, 0, 48.14, -42.34], [9E9, 9E9, 9E9, 9E9, 9E9, 9E9]];
	VAR jointtarget CDP_297 := [[11.5, 36.11, 5.72, 0, 48.17, -40.11], [9E9, 9E9, 9E9, 9E9, 9E9, 9E9]];
	VAR jointtarget CDP_298 := [[11.53, 36.15, 5.64, 0, 48.21, -37.88], [9E9, 9E9, 9E9, 9E9, 9E9, 9E9]];
	VAR jointtarget CDP_299 := [[11.57, 36.2, 5.56, 0, 48.24, -35.65], [9E9, 9E9, 9E9, 9E9, 9E9, 9E9]];
	VAR jointtarget CDP_300 := [[11.59, 36.23, 5.5, 0, 48.26, -34.54], [9E9, 9E9, 9E9, 9E9, 9E9, 9E9]];
	VAR jointtarget CDP_301 := [[11.6, 36.26, 5.45, 0, 48.28, -34.52], [9E9, 9E9, 9E9, 9E9, 9E9, 9E9]];
	VAR jointtarget CDP_302 := [[11.62, 36.29, 5.4, 0, 48.31, -34.5], [9E9, 9E9, 9E9, 9E9, 9E9, 9E9]];
	VAR jointtarget CDP_303 := [[11.64, 36.32, 5.35, 0, 48.33, -34.48], [9E9, 9E9, 9E9, 9E9, 9E9, 9E9]];
	VAR jointtarget CDP_304 := [[11.66, 36.35, 5.3, 0, 48.35, -34.46], [9E9, 9E9, 9E9, 9E9, 9E9, 9E9]];
	VAR jointtarget CDP_305 := [[11.68, 36.38, 5.25, 0, 48.37, -34.44], [9E9, 9E9, 9E9, 9E9, 9E9, 9E9]];
	VAR jointtarget CDP_306 := [[11.7, 36.41, 5.19, 0, 48.39, -34.42], [9E9, 9E9, 9E9, 9E9, 9E9, 9E9]];
	VAR jointtarget CDP_307 := [[11.72, 36.44, 5.14, 0, 48.41, -34.41], [9E9, 9E9, 9E9, 9E9, 9E9, 9E9]];
	VAR jointtarget CDP_308 := [[11.74, 36.47, 5.09, 0, 48.44, -34.39], [9E9, 9E9, 9E9, 9E9, 9E9, 9E9]];
	VAR jointtarget CDP_309 := [[11.76, 36.5, 5.04, 0, 48.46, -34.37], [9E9, 9E9, 9E9, 9E9, 9E9, 9E9]];
	VAR jointtarget CDP_310 := [[11.77, 36.53, 4.99, 0, 48.48, -34.35], [9E9, 9E9, 9E9, 9E9, 9E9, 9E9]];
	VAR jointtarget CDP_311 := [[11.79, 36.56, 4.93, 0, 48.5, -34.33], [9E9, 9E9, 9E9, 9E9, 9E9, 9E9]];
	VAR jointtarget CDP_312 := [[11.81, 36.59, 4.88, 0, 48.52, -34.31], [9E9, 9E9, 9E9, 9E9, 9E9, 9E9]];
	VAR jointtarget CDP_313 := [[11.83, 36.62, 4.83, 0, 48.54, -34.29], [9E9, 9E9, 9E9, 9E9, 9E9, 9E9]];
	VAR jointtarget CDP_314 := [[11.85, 36.66, 4.78, 0, 48.57, -34.27], [9E9, 9E9, 9E9, 9E9, 9E9, 9E9]];
	VAR jointtarget CDP_315 := [[11.87, 36.69, 4.73, 0, 48.59, -34.26], [9E9, 9E9, 9E9, 9E9, 9E9, 9E9]];
	VAR jointtarget CDP_316 := [[11.89, 36.72, 4.67, 0, 48.61, -34.24], [9E9, 9E9, 9E9, 9E9, 9E9, 9E9]];
	VAR jointtarget CDP_317 := [[11.91, 36.75, 4.62, 0, 48.63, -34.22], [9E9, 9E9, 9E9, 9E9, 9E9, 9E9]];
	VAR jointtarget CDP_318 := [[11.92, 36.78, 4.57, 0, 48.65, -34.2], [9E9, 9E9, 9E9, 9E9, 9E9, 9E9]];
	VAR jointtarget CDP_319 := [[11.94, 36.81, 4.52, 0, 48.68, -34.18], [9E9, 9E9, 9E9, 9E9, 9E9, 9E9]];
	VAR jointtarget CDP_320 := [[12.05, 36.94, 4.28, 0, 48.77, -40.77], [9E9, 9E9, 9E9, 9E9, 9E9, 9E9]];
	VAR jointtarget CDP_321 := [[12.18, 37.05, 4.1, 0, 48.85, -54.03], [9E9, 9E9, 9E9, 9E9, 9E9, 9E9]];
	VAR jointtarget CDP_322 := [[12.33, 37.12, 3.98, 0, 48.9, -67.26], [9E9, 9E9, 9E9, 9E9, 9E9, 9E9]];
	VAR jointtarget CDP_323 := [[12.49, 37.15, 3.93, 0, 48.92, -80.49], [9E9, 9E9, 9E9, 9E9, 9E9, 9E9]];
	VAR jointtarget CDP_324 := [[12.65, 37.13, 3.95, 0, 48.91, -93.72], [9E9, 9E9, 9E9, 9E9, 9E9, 9E9]];
	VAR jointtarget CDP_325 := [[12.8, 37.08, 4.04, 0, 48.88, -106.95], [9E9, 9E9, 9E9, 9E9, 9E9, 9E9]];
	VAR jointtarget CDP_326 := [[12.94, 36.99, 4.2, 0, 48.81, -120.2], [9E9, 9E9, 9E9, 9E9, 9E9, 9E9]];
	VAR jointtarget CDP_327 := [[13.06, 36.87, 4.41, 0, 48.72, -133.47], [9E9, 9E9, 9E9, 9E9, 9E9, 9E9]];
	VAR jointtarget CDP_328 := [[13.15, 36.72, 4.67, 0, 48.61, -146.77], [9E9, 9E9, 9E9, 9E9, 9E9, 9E9]];
	VAR jointtarget CDP_329 := [[13.2, 36.55, 4.96, 0, 48.49, -160.1], [9E9, 9E9, 9E9, 9E9, 9E9, 9E9]];
	VAR jointtarget CDP_330 := [[13.22, 36.37, 5.27, 0, 48.36, -173.47], [9E9, 9E9, 9E9, 9E9, 9E9, 9E9]];
	VAR jointtarget CDP_331 := [[13.2, 36.19, 5.57, 0, 48.24, -186.88], [9E9, 9E9, 9E9, 9E9, 9E9, 9E9]];
	VAR jointtarget CDP_332 := [[13.15, 36.03, 5.86, 0, 48.12, -200.32], [9E9, 9E9, 9E9, 9E9, 9E9, 9E9]];
	VAR jointtarget CDP_333 := [[13.06, 35.88, 6.11, 0, 48.01, -213.8], [9E9, 9E9, 9E9, 9E9, 9E9, 9E9]];
	VAR jointtarget CDP_334 := [[12.93, 35.76, 6.32, 0, 47.92, -227.31], [9E9, 9E9, 9E9, 9E9, 9E9, 9E9]];
	VAR jointtarget CDP_335 := [[12.79, 35.67, 6.47, 0, 47.86, -240.84], [9E9, 9E9, 9E9, 9E9, 9E9, 9E9]];
	VAR jointtarget CDP_336 := [[12.63, 35.62, 6.55, 0, 47.83, -254.39], [9E9, 9E9, 9E9, 9E9, 9E9, 9E9]];
	VAR jointtarget CDP_337 := [[12.47, 35.62, 6.56, 0, 47.82, -267.94], [9E9, 9E9, 9E9, 9E9, 9E9, 9E9]];
	VAR jointtarget CDP_338 := [[12.3, 35.65, 6.5, 0, 47.85, -281.49], [9E9, 9E9, 9E9, 9E9, 9E9, 9E9]];
	VAR jointtarget CDP_339 := [[12.15, 35.73, 6.37, 0, 47.9, -295.03], [9E9, 9E9, 9E9, 9E9, 9E9, 9E9]];
	VAR jointtarget CDP_340 := [[12.13, 35.75, 6.34, 0, 47.91, -301.75], [9E9, 9E9, 9E9, 9E9, 9E9, 9E9]];
	VAR jointtarget CDP_341 := [[12.1, 35.77, 6.31, 0, 47.93, -301.78], [9E9, 9E9, 9E9, 9E9, 9E9, 9E9]];
	VAR jointtarget CDP_342 := [[12.07, 35.79, 6.27, 0, 47.94, -301.81], [9E9, 9E9, 9E9, 9E9, 9E9, 9E9]];
	VAR jointtarget CDP_343 := [[12.04, 35.8, 6.24, 0, 47.96, -301.84], [9E9, 9E9, 9E9, 9E9, 9E9, 9E9]];
	VAR jointtarget CDP_344 := [[12.01, 35.82, 6.21, 0, 47.97, -301.87], [9E9, 9E9, 9E9, 9E9, 9E9, 9E9]];
	VAR jointtarget CDP_345 := [[11.98, 35.84, 6.17, 0, 47.98, -301.89], [9E9, 9E9, 9E9, 9E9, 9E9, 9E9]];
	VAR jointtarget CDP_346 := [[11.95, 35.86, 6.14, 0, 48, -301.92], [9E9, 9E9, 9E9, 9E9, 9E9, 9E9]];
	VAR jointtarget CDP_347 := [[11.92, 35.88, 6.11, 0, 48.01, -301.95], [9E9, 9E9, 9E9, 9E9, 9E9, 9E9]];
	VAR jointtarget CDP_348 := [[11.9, 35.9, 6.08, 0, 48.02, -301.98], [9E9, 9E9, 9E9, 9E9, 9E9, 9E9]];
	VAR jointtarget CDP_349 := [[11.87, 35.92, 6.04, 0, 48.04, -302.01], [9E9, 9E9, 9E9, 9E9, 9E9, 9E9]];
	VAR jointtarget CDP_350 := [[11.84, 35.94, 6.01, 0, 48.05, -302.04], [9E9, 9E9, 9E9, 9E9, 9E9, 9E9]];
	VAR jointtarget CDP_351 := [[11.81, 35.96, 5.98, 0, 48.07, -302.07], [9E9, 9E9, 9E9, 9E9, 9E9, 9E9]];
	VAR jointtarget CDP_352 := [[11.78, 35.98, 5.94, 0, 48.08, -302.09], [9E9, 9E9, 9E9, 9E9, 9E9, 9E9]];
	VAR jointtarget CDP_353 := [[11.75, 36, 5.91, 0, 48.09, -302.12], [9E9, 9E9, 9E9, 9E9, 9E9, 9E9]];
	VAR jointtarget CDP_354 := [[11.73, 36.02, 5.88, 0, 48.11, -302.15], [9E9, 9E9, 9E9, 9E9, 9E9, 9E9]];
	VAR jointtarget CDP_355 := [[11.7, 36.04, 5.84, 0, 48.12, -302.18], [9E9, 9E9, 9E9, 9E9, 9E9, 9E9]];
	VAR jointtarget CDP_356 := [[11.67, 36.06, 5.81, 0, 48.13, -302.21], [9E9, 9E9, 9E9, 9E9, 9E9, 9E9]];
	VAR jointtarget CDP_357 := [[11.64, 36.07, 5.78, 0, 48.15, -302.24], [9E9, 9E9, 9E9, 9E9, 9E9, 9E9]];
	VAR jointtarget CDP_358 := [[11.61, 36.09, 5.74, 0, 48.16, -302.27], [9E9, 9E9, 9E9, 9E9, 9E9, 9E9]];
	VAR jointtarget CDP_359 := [[11.58, 36.11, 5.71, 0, 48.18, -302.29], [9E9, 9E9, 9E9, 9E9, 9E9, 9E9]];
	VAR jointtarget CDP_360 := [[11.54, 36.14, 5.66, 0, 48.2, -301.24], [9E9, 9E9, 9E9, 9E9, 9E9, 9E9]];
	VAR jointtarget CDP_361 := [[11.49, 36.17, 5.61, 0, 48.22, -299.1], [9E9, 9E9, 9E9, 9E9, 9E9, 9E9]];
	VAR jointtarget CDP_362 := [[11.44, 36.2, 5.56, 0, 48.24, -296.95], [9E9, 9E9, 9E9, 9E9, 9E9, 9E9]];
	VAR jointtarget CDP_363 := [[11.39, 36.23, 5.52, 0, 48.26, -294.81], [9E9, 9E9, 9E9, 9E9, 9E9, 9E9]];
	VAR jointtarget CDP_364 := [[11.34, 36.25, 5.48, 0, 48.27, -292.67], [9E9, 9E9, 9E9, 9E9, 9E9, 9E9]];
	VAR jointtarget CDP_365 := [[11.28, 36.27, 5.44, 0, 48.29, -290.53], [9E9, 9E9, 9E9, 9E9, 9E9, 9E9]];
	VAR jointtarget CDP_366 := [[11.23, 36.29, 5.41, 0, 48.3, -288.38], [9E9, 9E9, 9E9, 9E9, 9E9, 9E9]];
	VAR jointtarget CDP_367 := [[11.18, 36.31, 5.38, 0, 48.32, -286.24], [9E9, 9E9, 9E9, 9E9, 9E9, 9E9]];
	VAR jointtarget CDP_368 := [[11.13, 36.32, 5.35, 0, 48.33, -284.1], [9E9, 9E9, 9E9, 9E9, 9E9, 9E9]];
	VAR jointtarget CDP_369 := [[11.07, 36.33, 5.33, 0, 48.33, -281.96], [9E9, 9E9, 9E9, 9E9, 9E9, 9E9]];
	VAR jointtarget CDP_370 := [[11.02, 36.34, 5.31, 0, 48.34, -279.82], [9E9, 9E9, 9E9, 9E9, 9E9, 9E9]];
	VAR jointtarget CDP_371 := [[10.96, 36.35, 5.3, 0, 48.35, -277.69], [9E9, 9E9, 9E9, 9E9, 9E9, 9E9]];
	VAR jointtarget CDP_372 := [[10.91, 36.36, 5.29, 0, 48.35, -275.55], [9E9, 9E9, 9E9, 9E9, 9E9, 9E9]];
	VAR jointtarget CDP_373 := [[10.85, 36.36, 5.28, 0, 48.35, -273.41], [9E9, 9E9, 9E9, 9E9, 9E9, 9E9]];
	VAR jointtarget CDP_374 := [[10.8, 36.36, 5.28, 0, 48.36, -271.27], [9E9, 9E9, 9E9, 9E9, 9E9, 9E9]];
	VAR jointtarget CDP_375 := [[10.74, 36.36, 5.28, 0, 48.36, -269.13], [9E9, 9E9, 9E9, 9E9, 9E9, 9E9]];
	VAR jointtarget CDP_376 := [[10.69, 36.36, 5.29, 0, 48.35, -266.99], [9E9, 9E9, 9E9, 9E9, 9E9, 9E9]];
	VAR jointtarget CDP_377 := [[10.63, 36.35, 5.3, 0, 48.35, -264.85], [9E9, 9E9, 9E9, 9E9, 9E9, 9E9]];
	VAR jointtarget CDP_378 := [[10.58, 36.35, 5.31, 0, 48.34, -262.71], [9E9, 9E9, 9E9, 9E9, 9E9, 9E9]];
	VAR jointtarget CDP_379 := [[10.52, 36.34, 5.33, 0, 48.34, -260.58], [9E9, 9E9, 9E9, 9E9, 9E9, 9E9]];
	VAR jointtarget CDP_380 := [[9.44, 36.13, 5.68, 0, 48.19, -260.56], [9E9, 9E9, 9E9, 9E9, 9E9, 9E9]];
	VAR jointtarget CDP_381 := [[8.36, 35.95, 6, 0, 48.06, -261.64], [9E9, 9E9, 9E9, 9E9, 9E9, 9E9]];
	VAR jointtarget CDP_382 := [[7.27, 35.78, 6.28, 0, 47.94, -262.73], [9E9, 9E9, 9E9, 9E9, 9E9, 9E9]];
	VAR jointtarget CDP_383 := [[6.17, 35.65, 6.51, 0, 47.84, -263.83], [9E9, 9E9, 9E9, 9E9, 9E9, 9E9]];
	VAR jointtarget CDP_384 := [[5.07, 35.53, 6.71, 0, 47.76, -264.93], [9E9, 9E9, 9E9, 9E9, 9E9, 9E9]];
	VAR jointtarget CDP_385 := [[3.97, 35.44, 6.87, 0, 47.69, -266.03], [9E9, 9E9, 9E9, 9E9, 9E9, 9E9]];
	VAR jointtarget CDP_386 := [[2.86, 35.37, 6.99, 0, 47.64, -267.14], [9E9, 9E9, 9E9, 9E9, 9E9, 9E9]];
	VAR jointtarget CDP_387 := [[1.75, 35.32, 7.07, 0, 47.61, -268.25], [9E9, 9E9, 9E9, 9E9, 9E9, 9E9]];
	VAR jointtarget CDP_388 := [[0.64, 35.29, 7.12, 0, 47.59, -269.36], [9E9, 9E9, 9E9, 9E9, 9E9, 9E9]];
	VAR jointtarget CDP_389 := [[-0.47, 35.29, 7.12, 0, 47.59, -270.47], [9E9, 9E9, 9E9, 9E9, 9E9, 9E9]];
	VAR jointtarget CDP_390 := [[-1.58, 35.31, 7.08, 0, 47.61, -271.58], [9E9, 9E9, 9E9, 9E9, 9E9, 9E9]];
	VAR jointtarget CDP_391 := [[-2.69, 35.36, 7.01, 0, 47.64, -272.69], [9E9, 9E9, 9E9, 9E9, 9E9, 9E9]];
	VAR jointtarget CDP_392 := [[-3.8, 35.42, 6.89, 0, 47.68, -273.8], [9E9, 9E9, 9E9, 9E9, 9E9, 9E9]];
	VAR jointtarget CDP_393 := [[-4.9, 35.51, 6.74, 0, 47.75, -274.9], [9E9, 9E9, 9E9, 9E9, 9E9, 9E9]];
	VAR jointtarget CDP_394 := [[-6, 35.63, 6.55, 0, 47.83, -276], [9E9, 9E9, 9E9, 9E9, 9E9, 9E9]];
	VAR jointtarget CDP_395 := [[-7.1, 35.76, 6.31, 0, 47.92, -277.1], [9E9, 9E9, 9E9, 9E9, 9E9, 9E9]];
	VAR jointtarget CDP_396 := [[-8.19, 35.92, 6.04, 0, 48.04, -278.19], [9E9, 9E9, 9E9, 9E9, 9E9, 9E9]];
	VAR jointtarget CDP_397 := [[-9.28, 36.1, 5.73, 0, 48.17, -279.28], [9E9, 9E9, 9E9, 9E9, 9E9, 9E9]];
	VAR jointtarget CDP_398 := [[-10.36, 36.3, 5.38, 0, 48.31, -280.36], [9E9, 9E9, 9E9, 9E9, 9E9, 9E9]];
	VAR jointtarget CDP_399 := [[-11.43, 36.53, 5, 0, 48.47, -281.43], [9E9, 9E9, 9E9, 9E9, 9E9, 9E9]];
	VAR jointtarget CDP_400 := [[-11.44, 36.53, 4.99, 0, 48.48, -281.78], [9E9, 9E9, 9E9, 9E9, 9E9, 9E9]];
	VAR jointtarget CDP_401 := [[-11.46, 36.54, 4.98, 0, 48.48, -282.45], [9E9, 9E9, 9E9, 9E9, 9E9, 9E9]];
	VAR jointtarget CDP_402 := [[-11.48, 36.54, 4.98, 0, 48.48, -283.13], [9E9, 9E9, 9E9, 9E9, 9E9, 9E9]];
	VAR jointtarget CDP_403 := [[-11.49, 36.54, 4.97, 0, 48.49, -283.81], [9E9, 9E9, 9E9, 9E9, 9E9, 9E9]];
	VAR jointtarget CDP_404 := [[-11.51, 36.55, 4.96, 0, 48.49, -284.49], [9E9, 9E9, 9E9, 9E9, 9E9, 9E9]];
	VAR jointtarget CDP_405 := [[-11.53, 36.55, 4.95, 0, 48.49, -285.17], [9E9, 9E9, 9E9, 9E9, 9E9, 9E9]];
	VAR jointtarget CDP_406 := [[-11.54, 36.56, 4.94, 0, 48.5, -285.84], [9E9, 9E9, 9E9, 9E9, 9E9, 9E9]];
	VAR jointtarget CDP_407 := [[-11.56, 36.56, 4.94, 0, 48.5, -286.52], [9E9, 9E9, 9E9, 9E9, 9E9, 9E9]];
	VAR jointtarget CDP_408 := [[-11.57, 36.57, 4.93, 0, 48.5, -287.2], [9E9, 9E9, 9E9, 9E9, 9E9, 9E9]];
	VAR jointtarget CDP_409 := [[-11.59, 36.57, 4.92, 0, 48.51, -287.88], [9E9, 9E9, 9E9, 9E9, 9E9, 9E9]];
	VAR jointtarget CDP_410 := [[-11.6, 36.58, 4.91, 0, 48.51, -288.56], [9E9, 9E9, 9E9, 9E9, 9E9, 9E9]];
	VAR jointtarget CDP_411 := [[-11.62, 36.59, 4.9, 0, 48.52, -289.23], [9E9, 9E9, 9E9, 9E9, 9E9, 9E9]];
	VAR jointtarget CDP_412 := [[-11.64, 36.59, 4.89, 0, 48.52, -289.91], [9E9, 9E9, 9E9, 9E9, 9E9, 9E9]];
	VAR jointtarget CDP_413 := [[-11.65, 36.6, 4.87, 0, 48.53, -290.59], [9E9, 9E9, 9E9, 9E9, 9E9, 9E9]];
	VAR jointtarget CDP_414 := [[-11.67, 36.61, 4.86, 0, 48.53, -291.27], [9E9, 9E9, 9E9, 9E9, 9E9, 9E9]];
	VAR jointtarget CDP_415 := [[-11.68, 36.61, 4.85, 0, 48.54, -291.94], [9E9, 9E9, 9E9, 9E9, 9E9, 9E9]];
	VAR jointtarget CDP_416 := [[-11.7, 36.62, 4.84, 0, 48.54, -292.62], [9E9, 9E9, 9E9, 9E9, 9E9, 9E9]];
	VAR jointtarget CDP_417 := [[-11.71, 36.63, 4.83, 0, 48.55, -293.3], [9E9, 9E9, 9E9, 9E9, 9E9, 9E9]];
	VAR jointtarget CDP_418 := [[-11.73, 36.63, 4.81, 0, 48.55, -293.98], [9E9, 9E9, 9E9, 9E9, 9E9, 9E9]];
	VAR jointtarget CDP_419 := [[-11.74, 36.64, 4.8, 0, 48.56, -294.65], [9E9, 9E9, 9E9, 9E9, 9E9, 9E9]];
	VAR jointtarget CDP_420 := [[-11.8, 36.67, 4.75, 0, 48.58, -295.04], [9E9, 9E9, 9E9, 9E9, 9E9, 9E9]];
	VAR jointtarget CDP_421 := [[-11.86, 36.7, 4.69, 0, 48.6, -295.11], [9E9, 9E9, 9E9, 9E9, 9E9, 9E9]];
	VAR jointtarget CDP_422 := [[-11.93, 36.74, 4.64, 0, 48.62, -295.17], [9E9, 9E9, 9E9, 9E9, 9E9, 9E9]];
	VAR jointtarget CDP_423 := [[-11.99, 36.77, 4.59, 0, 48.65, -295.23], [9E9, 9E9, 9E9, 9E9, 9E9, 9E9]];
	VAR jointtarget CDP_424 := [[-12.05, 36.8, 4.53, 0, 48.67, -295.29], [9E9, 9E9, 9E9, 9E9, 9E9, 9E9]];
	VAR jointtarget CDP_425 := [[-12.11, 36.83, 4.48, 0, 48.69, -295.35], [9E9, 9E9, 9E9, 9E9, 9E9, 9E9]];
	VAR jointtarget CDP_426 := [[-12.17, 36.86, 4.42, 0, 48.72, -295.41], [9E9, 9E9, 9E9, 9E9, 9E9, 9E9]];
	VAR jointtarget CDP_427 := [[-12.23, 36.89, 4.37, 0, 48.74, -295.47], [9E9, 9E9, 9E9, 9E9, 9E9, 9E9]];
	VAR jointtarget CDP_428 := [[-12.29, 36.92, 4.31, 0, 48.76, -295.53], [9E9, 9E9, 9E9, 9E9, 9E9, 9E9]];
	VAR jointtarget CDP_429 := [[-12.35, 36.96, 4.26, 0, 48.78, -295.59], [9E9, 9E9, 9E9, 9E9, 9E9, 9E9]];
	VAR jointtarget CDP_430 := [[-12.41, 36.99, 4.2, 0, 48.81, -295.65], [9E9, 9E9, 9E9, 9E9, 9E9, 9E9]];
	VAR jointtarget CDP_431 := [[-12.47, 37.02, 4.15, 0, 48.83, -295.71], [9E9, 9E9, 9E9, 9E9, 9E9, 9E9]];
	VAR jointtarget CDP_432 := [[-12.53, 37.05, 4.09, 0, 48.85, -295.77], [9E9, 9E9, 9E9, 9E9, 9E9, 9E9]];
	VAR jointtarget CDP_433 := [[-12.59, 37.08, 4.04, 0, 48.88, -295.83], [9E9, 9E9, 9E9, 9E9, 9E9, 9E9]];
	VAR jointtarget CDP_434 := [[-12.65, 37.12, 3.98, 0, 48.9, -295.89], [9E9, 9E9, 9E9, 9E9, 9E9, 9E9]];
	VAR jointtarget CDP_435 := [[-12.71, 37.15, 3.93, 0, 48.92, -295.95], [9E9, 9E9, 9E9, 9E9, 9E9, 9E9]];
	VAR jointtarget CDP_436 := [[-12.77, 37.18, 3.87, 0, 48.95, -296.01], [9E9, 9E9, 9E9, 9E9, 9E9, 9E9]];
	VAR jointtarget CDP_437 := [[-12.83, 37.21, 3.81, 0, 48.97, -296.07], [9E9, 9E9, 9E9, 9E9, 9E9, 9E9]];
	VAR jointtarget CDP_438 := [[-12.89, 37.25, 3.76, 0, 49, -296.13], [9E9, 9E9, 9E9, 9E9, 9E9, 9E9]];
	VAR jointtarget CDP_439 := [[-12.95, 37.28, 3.7, 0, 49.02, -296.19], [9E9, 9E9, 9E9, 9E9, 9E9, 9E9]];
	VAR jointtarget CDP_440 := [[-13.07, 37.33, 3.61, 0, 49.06, -291.14], [9E9, 9E9, 9E9, 9E9, 9E9, 9E9]];
	VAR jointtarget CDP_441 := [[-13.19, 37.36, 3.56, 0, 49.08, -280.95], [9E9, 9E9, 9E9, 9E9, 9E9, 9E9]];
	VAR jointtarget CDP_442 := [[-13.32, 37.36, 3.56, 0, 49.08, -270.75], [9E9, 9E9, 9E9, 9E9, 9E9, 9E9]];
	VAR jointtarget CDP_443 := [[-13.45, 37.34, 3.6, 0, 49.06, -260.55], [9E9, 9E9, 9E9, 9E9, 9E9, 9E9]];
	VAR jointtarget CDP_444 := [[-13.57, 37.29, 3.69, 0, 49.03, -250.35], [9E9, 9E9, 9E9, 9E9, 9E9, 9E9]];
	VAR jointtarget CDP_445 := [[-13.68, 37.22, 3.81, 0, 48.97, -240.14], [9E9, 9E9, 9E9, 9E9, 9E9, 9E9]];
	VAR jointtarget CDP_446 := [[-13.78, 37.12, 3.97, 0, 48.91, -229.91], [9E9, 9E9, 9E9, 9E9, 9E9, 9E9]];
	VAR jointtarget CDP_447 := [[-13.86, 37.01, 4.16, 0, 48.83, -219.67], [9E9, 9E9, 9E9, 9E9, 9E9, 9E9]];
	VAR jointtarget CDP_448 := [[-13.93, 36.89, 4.38, 0, 48.73, -209.41], [9E9, 9E9, 9E9, 9E9, 9E9, 9E9]];
	VAR jointtarget CDP_449 := [[-13.97, 36.75, 4.61, 0, 48.64, -199.13], [9E9, 9E9, 9E9, 9E9, 9E9, 9E9]];
	VAR jointtarget CDP_450 := [[-13.99, 36.61, 4.85, 0, 48.53, -188.83], [9E9, 9E9, 9E9, 9E9, 9E9, 9E9]];
	VAR jointtarget CDP_451 := [[-13.98, 36.47, 5.1, 0, 48.43, -178.5], [9E9, 9E9, 9E9, 9E9, 9E9, 9E9]];
	VAR jointtarget CDP_452 := [[-13.96, 36.33, 5.34, 0, 48.33, -168.15], [9E9, 9E9, 9E9, 9E9, 9E9, 9E9]];
	VAR jointtarget CDP_453 := [[-13.91, 36.2, 5.57, 0, 48.24, -157.77], [9E9, 9E9, 9E9, 9E9, 9E9, 9E9]];
	VAR jointtarget CDP_454 := [[-13.84, 36.08, 5.77, 0, 48.15, -147.38], [9E9, 9E9, 9E9, 9E9, 9E9, 9E9]];
	VAR jointtarget CDP_455 := [[-13.75, 35.97, 5.95, 0, 48.08, -136.97], [9E9, 9E9, 9E9, 9E9, 9E9, 9E9]];
	VAR jointtarget CDP_456 := [[-13.64, 35.89, 6.1, 0, 48.01, -126.54], [9E9, 9E9, 9E9, 9E9, 9E9, 9E9]];
	VAR jointtarget CDP_457 := [[-13.52, 35.82, 6.21, 0, 47.97, -116.09], [9E9, 9E9, 9E9, 9E9, 9E9, 9E9]];
	VAR jointtarget CDP_458 := [[-13.4, 35.79, 6.27, 0, 47.94, -105.64], [9E9, 9E9, 9E9, 9E9, 9E9, 9E9]];
	VAR jointtarget CDP_459 := [[-13.27, 35.77, 6.29, 0, 47.93, -95.19], [9E9, 9E9, 9E9, 9E9, 9E9, 9E9]];
	VAR jointtarget CDP_460 := [[-13.2, 35.77, 6.29, 0, 47.93, -89.96], [9E9, 9E9, 9E9, 9E9, 9E9, 9E9]];
	VAR jointtarget CDP_461 := [[-13.13, 35.77, 6.29, 0, 47.93, -89.89], [9E9, 9E9, 9E9, 9E9, 9E9, 9E9]];
	VAR jointtarget CDP_462 := [[-13.06, 35.77, 6.29, 0, 47.94, -89.82], [9E9, 9E9, 9E9, 9E9, 9E9, 9E9]];
	VAR jointtarget CDP_463 := [[-12.99, 35.77, 6.29, 0, 47.94, -89.75], [9E9, 9E9, 9E9, 9E9, 9E9, 9E9]];
	VAR jointtarget CDP_464 := [[-12.93, 35.77, 6.29, 0, 47.94, -89.69], [9E9, 9E9, 9E9, 9E9, 9E9, 9E9]];
	VAR jointtarget CDP_465 := [[-12.86, 35.77, 6.29, 0, 47.94, -89.62], [9E9, 9E9, 9E9, 9E9, 9E9, 9E9]];
	VAR jointtarget CDP_466 := [[-12.79, 35.77, 6.29, 0, 47.94, -89.55], [9E9, 9E9, 9E9, 9E9, 9E9, 9E9]];
	VAR jointtarget CDP_467 := [[-12.72, 35.77, 6.29, 0, 47.94, -89.48], [9E9, 9E9, 9E9, 9E9, 9E9, 9E9]];
	VAR jointtarget CDP_468 := [[-12.65, 35.77, 6.29, 0, 47.94, -89.41], [9E9, 9E9, 9E9, 9E9, 9E9, 9E9]];
	VAR jointtarget CDP_469 := [[-12.59, 35.77, 6.29, 0, 47.94, -89.35], [9E9, 9E9, 9E9, 9E9, 9E9, 9E9]];
	VAR jointtarget CDP_470 := [[-12.52, 35.77, 6.28, 0, 47.94, -89.28], [9E9, 9E9, 9E9, 9E9, 9E9, 9E9]];
	VAR jointtarget CDP_471 := [[-12.45, 35.77, 6.28, 0, 47.95, -89.21], [9E9, 9E9, 9E9, 9E9, 9E9, 9E9]];
	VAR jointtarget CDP_472 := [[-12.38, 35.77, 6.28, 0, 47.95, -89.14], [9E9, 9E9, 9E9, 9E9, 9E9, 9E9]];
	VAR jointtarget CDP_473 := [[-12.32, 35.77, 6.28, 0, 47.95, -89.07], [9E9, 9E9, 9E9, 9E9, 9E9, 9E9]];
	VAR jointtarget CDP_474 := [[-12.25, 35.77, 6.28, 0, 47.95, -89.01], [9E9, 9E9, 9E9, 9E9, 9E9, 9E9]];
	VAR jointtarget CDP_475 := [[-12.18, 35.77, 6.27, 0, 47.95, -88.94], [9E9, 9E9, 9E9, 9E9, 9E9, 9E9]];
	VAR jointtarget CDP_476 := [[-12.11, 35.77, 6.27, 0, 47.95, -88.87], [9E9, 9E9, 9E9, 9E9, 9E9, 9E9]];
	VAR jointtarget CDP_477 := [[-12.04, 35.78, 6.27, 0, 47.96, -88.8], [9E9, 9E9, 9E9, 9E9, 9E9, 9E9]];
	VAR jointtarget CDP_478 := [[-11.98, 35.78, 6.27, 0, 47.96, -88.74], [9E9, 9E9, 9E9, 9E9, 9E9, 9E9]];
	VAR jointtarget CDP_479 := [[-11.91, 35.78, 6.26, 0, 47.96, -88.67], [9E9, 9E9, 9E9, 9E9, 9E9, 9E9]];
	VAR jointtarget CDP_480 := [[-11.89, 35.78, 6.26, 0, 47.96, -88.98], [9E9, 9E9, 9E9, 9E9, 9E9, 9E9]];
	VAR jointtarget CDP_481 := [[-11.87, 35.78, 6.26, 0, 47.96, -89.63], [9E9, 9E9, 9E9, 9E9, 9E9, 9E9]];
	VAR jointtarget CDP_482 := [[-11.86, 35.78, 6.26, 0, 47.96, -90.27], [9E9, 9E9, 9E9, 9E9, 9E9, 9E9]];
	VAR jointtarget CDP_483 := [[-11.84, 35.78, 6.26, 0, 47.96, -90.92], [9E9, 9E9, 9E9, 9E9, 9E9, 9E9]];
	VAR jointtarget CDP_484 := [[-11.82, 35.78, 6.26, 0, 47.96, -91.56], [9E9, 9E9, 9E9, 9E9, 9E9, 9E9]];
	VAR jointtarget CDP_485 := [[-11.81, 35.78, 6.27, 0, 47.96, -92.21], [9E9, 9E9, 9E9, 9E9, 9E9, 9E9]];
	VAR jointtarget CDP_486 := [[-11.79, 35.77, 6.27, 0, 47.96, -92.85], [9E9, 9E9, 9E9, 9E9, 9E9, 9E9]];
	VAR jointtarget CDP_487 := [[-11.77, 35.77, 6.27, 0, 47.96, -93.5], [9E9, 9E9, 9E9, 9E9, 9E9, 9E9]];
	VAR jointtarget CDP_488 := [[-11.76, 35.77, 6.27, 0, 47.96, -94.14], [9E9, 9E9, 9E9, 9E9, 9E9, 9E9]];
	VAR jointtarget CDP_489 := [[-11.74, 35.77, 6.27, 0, 47.96, -94.79], [9E9, 9E9, 9E9, 9E9, 9E9, 9E9]];
	VAR jointtarget CDP_490 := [[-11.72, 35.77, 6.28, 0, 47.95, -95.43], [9E9, 9E9, 9E9, 9E9, 9E9, 9E9]];
	VAR jointtarget CDP_491 := [[-11.71, 35.77, 6.28, 0, 47.95, -96.08], [9E9, 9E9, 9E9, 9E9, 9E9, 9E9]];
	VAR jointtarget CDP_492 := [[-11.69, 35.76, 6.28, 0, 47.95, -96.72], [9E9, 9E9, 9E9, 9E9, 9E9, 9E9]];
	VAR jointtarget CDP_493 := [[-11.67, 35.76, 6.29, 0, 47.95, -97.37], [9E9, 9E9, 9E9, 9E9, 9E9, 9E9]];
	VAR jointtarget CDP_494 := [[-11.66, 35.76, 6.29, 0, 47.95, -98.01], [9E9, 9E9, 9E9, 9E9, 9E9, 9E9]];
	VAR jointtarget CDP_495 := [[-11.64, 35.76, 6.3, 0, 47.95, -98.66], [9E9, 9E9, 9E9, 9E9, 9E9, 9E9]];
	VAR jointtarget CDP_496 := [[-11.62, 35.75, 6.3, 0, 47.94, -99.31], [9E9, 9E9, 9E9, 9E9, 9E9, 9E9]];
	VAR jointtarget CDP_497 := [[-11.61, 35.75, 6.31, 0, 47.94, -99.95], [9E9, 9E9, 9E9, 9E9, 9E9, 9E9]];
	VAR jointtarget CDP_498 := [[-11.59, 35.75, 6.31, 0, 47.94, -100.6], [9E9, 9E9, 9E9, 9E9, 9E9, 9E9]];
	VAR jointtarget CDP_499 := [[-11.57, 35.74, 6.32, 0, 47.94, -101.24], [9E9, 9E9, 9E9, 9E9, 9E9, 9E9]];
	VAR jointtarget CDP_500 := [[-10.48, 35.52, 6.71, 0, 47.77, -100.48], [9E9, 9E9, 9E9, 9E9, 9E9, 9E9]];
	VAR jointtarget CDP_501 := [[-9.38, 35.31, 7.06, 0, 47.63, -99.38], [9E9, 9E9, 9E9, 9E9, 9E9, 9E9]];
	VAR jointtarget CDP_502 := [[-8.27, 35.13, 7.37, 0, 47.5, -98.27], [9E9, 9E9, 9E9, 9E9, 9E9, 9E9]];
	VAR jointtarget CDP_503 := [[-7.15, 34.97, 7.65, 0, 47.39, -97.15], [9E9, 9E9, 9E9, 9E9, 9E9, 9E9]];
	VAR jointtarget CDP_504 := [[-6.03, 34.83, 7.88, 0, 47.29, -96.03], [9E9, 9E9, 9E9, 9E9, 9E9, 9E9]];
	VAR jointtarget CDP_505 := [[-4.9, 34.72, 8.07, 0, 47.21, -94.9], [9E9, 9E9, 9E9, 9E9, 9E9, 9E9]];
	VAR jointtarget CDP_506 := [[-3.77, 34.63, 8.23, 0, 47.15, -93.77], [9E9, 9E9, 9E9, 9E9, 9E9, 9E9]];
	VAR jointtarget CDP_507 := [[-2.64, 34.56, 8.34, 0, 47.1, -92.64], [9E9, 9E9, 9E9, 9E9, 9E9, 9E9]];
	VAR jointtarget CDP_508 := [[-1.51, 34.52, 8.41, 0, 47.07, -91.51], [9E9, 9E9, 9E9, 9E9, 9E9, 9E9]];
	VAR jointtarget CDP_509 := [[-0.37, 34.5, 8.44, 0, 47.06, -90.37], [9E9, 9E9, 9E9, 9E9, 9E9, 9E9]];
	VAR jointtarget CDP_510 := [[0.76, 34.5, 8.44, 0, 47.06, -89.24], [9E9, 9E9, 9E9, 9E9, 9E9, 9E9]];
	VAR jointtarget CDP_511 := [[1.9, 34.53, 8.39, 0, 47.08, -88.1], [9E9, 9E9, 9E9, 9E9, 9E9, 9E9]];
	VAR jointtarget CDP_512 := [[3.03, 34.58, 8.3, 0, 47.11, -86.97], [9E9, 9E9, 9E9, 9E9, 9E9, 9E9]];
	VAR jointtarget CDP_513 := [[4.16, 34.66, 8.18, 0, 47.17, -85.84], [9E9, 9E9, 9E9, 9E9, 9E9, 9E9]];
	VAR jointtarget CDP_514 := [[5.29, 34.75, 8.01, 0, 47.24, -84.71], [9E9, 9E9, 9E9, 9E9, 9E9, 9E9]];
	VAR jointtarget CDP_515 := [[6.42, 34.87, 7.8, 0, 47.32, -83.58], [9E9, 9E9, 9E9, 9E9, 9E9, 9E9]];
	VAR jointtarget CDP_516 := [[7.54, 35.02, 7.56, 0, 47.42, -82.46], [9E9, 9E9, 9E9, 9E9, 9E9, 9E9]];
	VAR jointtarget CDP_517 := [[8.65, 35.19, 7.27, 0, 47.54, -81.35], [9E9, 9E9, 9E9, 9E9, 9E9, 9E9]];
	VAR jointtarget CDP_518 := [[9.76, 35.38, 6.95, 0, 47.68, -80.24], [9E9, 9E9, 9E9, 9E9, 9E9, 9E9]];
	VAR jointtarget CDP_519 := [[10.86, 35.59, 6.58, 0, 47.83, -79.14], [9E9, 9E9, 9E9, 9E9, 9E9, 9E9]];
	VAR jointtarget CDP_520 := [[10.87, 35.59, 6.57, 0, 47.83, -79.46], [9E9, 9E9, 9E9, 9E9, 9E9, 9E9]];
	VAR jointtarget CDP_521 := [[10.89, 35.6, 6.57, 0, 47.83, -80.1], [9E9, 9E9, 9E9, 9E9, 9E9, 9E9]];
	VAR jointtarget CDP_522 := [[10.91, 35.6, 6.56, 0, 47.84, -80.75], [9E9, 9E9, 9E9, 9E9, 9E9, 9E9]];
	VAR jointtarget CDP_523 := [[10.92, 35.6, 6.56, 0, 47.84, -81.39], [9E9, 9E9, 9E9, 9E9, 9E9, 9E9]];
	VAR jointtarget CDP_524 := [[10.94, 35.61, 6.55, 0, 47.84, -82.04], [9E9, 9E9, 9E9, 9E9, 9E9, 9E9]];
	VAR jointtarget CDP_525 := [[10.96, 35.61, 6.55, 0, 47.84, -82.68], [9E9, 9E9, 9E9, 9E9, 9E9, 9E9]];
	VAR jointtarget CDP_526 := [[10.97, 35.61, 6.55, 0, 47.84, -83.33], [9E9, 9E9, 9E9, 9E9, 9E9, 9E9]];
	VAR jointtarget CDP_527 := [[10.99, 35.61, 6.54, 0, 47.84, -83.97], [9E9, 9E9, 9E9, 9E9, 9E9, 9E9]];
	VAR jointtarget CDP_528 := [[11.01, 35.61, 6.54, 0, 47.84, -84.62], [9E9, 9E9, 9E9, 9E9, 9E9, 9E9]];
	VAR jointtarget CDP_529 := [[11.02, 35.62, 6.54, 0, 47.85, -85.27], [9E9, 9E9, 9E9, 9E9, 9E9, 9E9]];
	VAR jointtarget CDP_530 := [[11.04, 35.62, 6.54, 0, 47.85, -85.91], [9E9, 9E9, 9E9, 9E9, 9E9, 9E9]];
	VAR jointtarget CDP_531 := [[11.06, 35.62, 6.53, 0, 47.85, -86.56], [9E9, 9E9, 9E9, 9E9, 9E9, 9E9]];
	VAR jointtarget CDP_532 := [[11.07, 35.62, 6.53, 0, 47.85, -87.2], [9E9, 9E9, 9E9, 9E9, 9E9, 9E9]];
	VAR jointtarget CDP_533 := [[11.09, 35.62, 6.53, 0, 47.85, -87.85], [9E9, 9E9, 9E9, 9E9, 9E9, 9E9]];
	VAR jointtarget CDP_534 := [[11.11, 35.62, 6.53, 0, 47.85, -88.49], [9E9, 9E9, 9E9, 9E9, 9E9, 9E9]];
	VAR jointtarget CDP_535 := [[11.13, 35.62, 6.53, 0, 47.85, -89.14], [9E9, 9E9, 9E9, 9E9, 9E9, 9E9]];
	VAR jointtarget CDP_536 := [[11.14, 35.62, 6.53, 0, 47.85, -89.78], [9E9, 9E9, 9E9, 9E9, 9E9, 9E9]];
	VAR jointtarget CDP_537 := [[11.16, 35.62, 6.53, 0, 47.85, -90.43], [9E9, 9E9, 9E9, 9E9, 9E9, 9E9]];
	VAR jointtarget CDP_538 := [[11.18, 35.62, 6.53, 0, 47.85, -91.07], [9E9, 9E9, 9E9, 9E9, 9E9, 9E9]];
	VAR jointtarget CDP_539 := [[11.19, 35.62, 6.53, 0, 47.85, -91.72], [9E9, 9E9, 9E9, 9E9, 9E9, 9E9]];
	VAR jointtarget CDP_540 := [[11.26, 35.62, 6.54, 0, 47.85, -91.98], [9E9, 9E9, 9E9, 9E9, 9E9, 9E9]];
	VAR jointtarget CDP_541 := [[11.33, 35.61, 6.54, 0, 47.85, -91.91], [9E9, 9E9, 9E9, 9E9, 9E9, 9E9]];
	VAR jointtarget CDP_542 := [[11.4, 35.61, 6.54, 0, 47.84, -91.84], [9E9, 9E9, 9E9, 9E9, 9E9, 9E9]];
	VAR jointtarget CDP_543 := [[11.47, 35.61, 6.55, 0, 47.84, -91.78], [9E9, 9E9, 9E9, 9E9, 9E9, 9E9]];
	VAR jointtarget CDP_544 := [[11.53, 35.61, 6.55, 0, 47.84, -91.71], [9E9, 9E9, 9E9, 9E9, 9E9, 9E9]];
	VAR jointtarget CDP_545 := [[11.6, 35.61, 6.56, 0, 47.84, -91.64], [9E9, 9E9, 9E9, 9E9, 9E9, 9E9]];
	VAR jointtarget CDP_546 := [[11.67, 35.6, 6.56, 0, 47.84, -91.57], [9E9, 9E9, 9E9, 9E9, 9E9, 9E9]];
	VAR jointtarget CDP_547 := [[11.74, 35.6, 6.56, 0, 47.84, -91.5], [9E9, 9E9, 9E9, 9E9, 9E9, 9E9]];
	VAR jointtarget CDP_548 := [[11.81, 35.6, 6.57, 0, 47.83, -91.44], [9E9, 9E9, 9E9, 9E9, 9E9, 9E9]];
	VAR jointtarget CDP_549 := [[11.87, 35.6, 6.57, 0, 47.83, -91.37], [9E9, 9E9, 9E9, 9E9, 9E9, 9E9]];
	VAR jointtarget CDP_550 := [[11.94, 35.6, 6.57, 0, 47.83, -91.3], [9E9, 9E9, 9E9, 9E9, 9E9, 9E9]];
	VAR jointtarget CDP_551 := [[12.01, 35.59, 6.58, 0, 47.83, -91.23], [9E9, 9E9, 9E9, 9E9, 9E9, 9E9]];
	VAR jointtarget CDP_552 := [[12.08, 35.59, 6.58, 0, 47.83, -91.16], [9E9, 9E9, 9E9, 9E9, 9E9, 9E9]];
	VAR jointtarget CDP_553 := [[12.15, 35.59, 6.58, 0, 47.83, -91.09], [9E9, 9E9, 9E9, 9E9, 9E9, 9E9]];
	VAR jointtarget CDP_554 := [[12.21, 35.59, 6.58, 0, 47.83, -91.03], [9E9, 9E9, 9E9, 9E9, 9E9, 9E9]];
	VAR jointtarget CDP_555 := [[12.28, 35.59, 6.58, 0, 47.83, -90.96], [9E9, 9E9, 9E9, 9E9, 9E9, 9E9]];
	VAR jointtarget CDP_556 := [[12.35, 35.59, 6.59, 0, 47.83, -90.89], [9E9, 9E9, 9E9, 9E9, 9E9, 9E9]];
	VAR jointtarget CDP_557 := [[12.42, 35.59, 6.59, 0, 47.83, -90.82], [9E9, 9E9, 9E9, 9E9, 9E9, 9E9]];
	VAR jointtarget CDP_558 := [[12.49, 35.59, 6.59, 0, 47.82, -90.75], [9E9, 9E9, 9E9, 9E9, 9E9, 9E9]];
	VAR jointtarget CDP_559 := [[12.55, 35.58, 6.59, 0, 47.82, -90.69], [9E9, 9E9, 9E9, 9E9, 9E9, 9E9]];
	VAR jointtarget CDP_560 := [[12.69, 35.6, 6.57, 0, 47.83, -85.39], [9E9, 9E9, 9E9, 9E9, 9E9, 9E9]];
	VAR jointtarget CDP_561 := [[12.81, 35.63, 6.51, 0, 47.86, -74.94], [9E9, 9E9, 9E9, 9E9, 9E9, 9E9]];
	VAR jointtarget CDP_562 := [[12.93, 35.69, 6.41, 0, 47.9, -64.5], [9E9, 9E9, 9E9, 9E9, 9E9, 9E9]];
	VAR jointtarget CDP_563 := [[13.04, 35.78, 6.26, 0, 47.96, -54.07], [9E9, 9E9, 9E9, 9E9, 9E9, 9E9]];
	VAR jointtarget CDP_564 := [[13.13, 35.88, 6.09, 0, 48.03, -43.65], [9E9, 9E9, 9E9, 9E9, 9E9, 9E9]];
	VAR jointtarget CDP_565 := [[13.2, 36, 5.88, 0, 48.12, -33.25], [9E9, 9E9, 9E9, 9E9, 9E9, 9E9]];
	VAR jointtarget CDP_566 := [[13.25, 36.13, 5.66, 0, 48.21, -22.88], [9E9, 9E9, 9E9, 9E9, 9E9, 9E9]];
	VAR jointtarget CDP_567 := [[13.28, 36.27, 5.42, 0, 48.31, -12.53], [9E9, 9E9, 9E9, 9E9, 9E9, 9E9]];
	VAR jointtarget CDP_568 := [[13.29, 36.41, 5.17, 0, 48.42, -2.2], [9E9, 9E9, 9E9, 9E9, 9E9, 9E9]];
	VAR jointtarget CDP_569 := [[13.27, 36.55, 4.93, 0, 48.52, 8.11], [9E9, 9E9, 9E9, 9E9, 9E9, 9E9]];
	VAR jointtarget CDP_570 := [[13.23, 36.69, 4.7, 0, 48.62, 18.39], [9E9, 9E9, 9E9, 9E9, 9E9, 9E9]];
	VAR jointtarget CDP_571 := [[13.17, 36.81, 4.48, 0, 48.71, 28.65], [9E9, 9E9, 9E9, 9E9, 9E9, 9E9]];
	VAR jointtarget CDP_572 := [[13.08, 36.93, 4.29, 0, 48.79, 38.9], [9E9, 9E9, 9E9, 9E9, 9E9, 9E9]];
	VAR jointtarget CDP_573 := [[12.99, 37.02, 4.12, 0, 48.86, 49.12], [9E9, 9E9, 9E9, 9E9, 9E9, 9E9]];
	VAR jointtarget CDP_574 := [[12.88, 37.09, 4, 0, 48.91, 59.33], [9E9, 9E9, 9E9, 9E9, 9E9, 9E9]];
	VAR jointtarget CDP_575 := [[12.75, 37.14, 3.91, 0, 48.94, 69.54], [9E9, 9E9, 9E9, 9E9, 9E9, 9E9]];
	VAR jointtarget CDP_576 := [[12.63, 37.17, 3.87, 0, 48.96, 79.73], [9E9, 9E9, 9E9, 9E9, 9E9, 9E9]];
	VAR jointtarget CDP_577 := [[12.5, 37.17, 3.87, 0, 48.96, 89.93], [9E9, 9E9, 9E9, 9E9, 9E9, 9E9]];
	VAR jointtarget CDP_578 := [[12.37, 37.14, 3.91, 0, 48.94, 100.13], [9E9, 9E9, 9E9, 9E9, 9E9, 9E9]];
	VAR jointtarget CDP_579 := [[12.25, 37.09, 4, 0, 48.91, 110.33], [9E9, 9E9, 9E9, 9E9, 9E9, 9E9]];
	VAR jointtarget CDP_580 := [[12.19, 37.06, 4.05, 0, 48.89, 115.43], [9E9, 9E9, 9E9, 9E9, 9E9, 9E9]];
	VAR jointtarget CDP_581 := [[12.13, 37.03, 4.11, 0, 48.86, 115.37], [9E9, 9E9, 9E9, 9E9, 9E9, 9E9]];
	VAR jointtarget CDP_582 := [[12.07, 37, 4.16, 0, 48.84, 115.31], [9E9, 9E9, 9E9, 9E9, 9E9, 9E9]];
	VAR jointtarget CDP_583 := [[12.01, 36.97, 4.22, 0, 48.82, 115.25], [9E9, 9E9, 9E9, 9E9, 9E9, 9E9]];
	VAR jointtarget CDP_584 := [[11.95, 36.94, 4.27, 0, 48.79, 115.19], [9E9, 9E9, 9E9, 9E9, 9E9, 9E9]];
	VAR jointtarget CDP_585 := [[11.89, 36.9, 4.33, 0, 48.77, 115.13], [9E9, 9E9, 9E9, 9E9, 9E9, 9E9]];
	VAR jointtarget CDP_586 := [[11.83, 36.87, 4.38, 0, 48.75, 115.07], [9E9, 9E9, 9E9, 9E9, 9E9, 9E9]];
	VAR jointtarget CDP_587 := [[11.77, 36.84, 4.43, 0, 48.73, 115.01], [9E9, 9E9, 9E9, 9E9, 9E9, 9E9]];
	VAR jointtarget CDP_588 := [[11.71, 36.81, 4.49, 0, 48.7, 114.95], [9E9, 9E9, 9E9, 9E9, 9E9, 9E9]];
	VAR jointtarget CDP_589 := [[11.65, 36.78, 4.54, 0, 48.68, 114.89], [9E9, 9E9, 9E9, 9E9, 9E9, 9E9]];
	VAR jointtarget CDP_590 := [[11.59, 36.75, 4.59, 0, 48.66, 114.83], [9E9, 9E9, 9E9, 9E9, 9E9, 9E9]];
	VAR jointtarget CDP_591 := [[11.53, 36.72, 4.65, 0, 48.64, 114.77], [9E9, 9E9, 9E9, 9E9, 9E9, 9E9]];
	VAR jointtarget CDP_592 := [[11.47, 36.69, 4.7, 0, 48.61, 114.71], [9E9, 9E9, 9E9, 9E9, 9E9, 9E9]];
	VAR jointtarget CDP_593 := [[11.4, 36.66, 4.75, 0, 48.59, 114.64], [9E9, 9E9, 9E9, 9E9, 9E9, 9E9]];
	VAR jointtarget CDP_594 := [[11.34, 36.62, 4.81, 0, 48.57, 114.58], [9E9, 9E9, 9E9, 9E9, 9E9, 9E9]];
	VAR jointtarget CDP_595 := [[11.28, 36.59, 4.86, 0, 48.55, 114.52], [9E9, 9E9, 9E9, 9E9, 9E9, 9E9]];
	VAR jointtarget CDP_596 := [[11.22, 36.56, 4.91, 0, 48.53, 114.46], [9E9, 9E9, 9E9, 9E9, 9E9, 9E9]];
	VAR jointtarget CDP_597 := [[11.16, 36.53, 4.96, 0, 48.5, 114.4], [9E9, 9E9, 9E9, 9E9, 9E9, 9E9]];
	VAR jointtarget CDP_598 := [[11.1, 36.5, 5.02, 0, 48.48, 114.34], [9E9, 9E9, 9E9, 9E9, 9E9, 9E9]];
	VAR jointtarget CDP_599 := [[11.04, 36.47, 5.07, 0, 48.46, 114.28], [9E9, 9E9, 9E9, 9E9, 9E9, 9E9]];
	VAR jointtarget CDP_600 := [[11.02, 36.47, 5.08, 0, 48.45, 113.93], [9E9, 9E9, 9E9, 9E9, 9E9, 9E9]];
	VAR jointtarget CDP_601 := [[11.01, 36.46, 5.09, 0, 48.45, 113.26], [9E9, 9E9, 9E9, 9E9, 9E9, 9E9]];
	VAR jointtarget CDP_602 := [[10.99, 36.45, 5.1, 0, 48.44, 112.58], [9E9, 9E9, 9E9, 9E9, 9E9, 9E9]];
	VAR jointtarget CDP_603 := [[10.98, 36.44, 5.12, 0, 48.44, 111.9], [9E9, 9E9, 9E9, 9E9, 9E9, 9E9]];
	VAR jointtarget CDP_604 := [[10.96, 36.44, 5.13, 0, 48.43, 111.22], [9E9, 9E9, 9E9, 9E9, 9E9, 9E9]];
	VAR jointtarget CDP_605 := [[10.95, 36.43, 5.14, 0, 48.43, 110.55], [9E9, 9E9, 9E9, 9E9, 9E9, 9E9]];
	VAR jointtarget CDP_606 := [[10.93, 36.43, 5.15, 0, 48.43, 109.87], [9E9, 9E9, 9E9, 9E9, 9E9, 9E9]];
	VAR jointtarget CDP_607 := [[10.91, 36.42, 5.16, 0, 48.42, 109.19], [9E9, 9E9, 9E9, 9E9, 9E9, 9E9]];
	VAR jointtarget CDP_608 := [[10.9, 36.41, 5.17, 0, 48.42, 108.51], [9E9, 9E9, 9E9, 9E9, 9E9, 9E9]];
	VAR jointtarget CDP_609 := [[10.88, 36.41, 5.18, 0, 48.41, 107.83], [9E9, 9E9, 9E9, 9E9, 9E9, 9E9]];
	VAR jointtarget CDP_610 := [[10.87, 36.4, 5.19, 0, 48.41, 107.16], [9E9, 9E9, 9E9, 9E9, 9E9, 9E9]];
	VAR jointtarget CDP_611 := [[10.85, 36.4, 5.2, 0, 48.41, 106.48], [9E9, 9E9, 9E9, 9E9, 9E9, 9E9]];
	VAR jointtarget CDP_612 := [[10.83, 36.39, 5.21, 0, 48.4, 105.8], [9E9, 9E9, 9E9, 9E9, 9E9, 9E9]];
	VAR jointtarget CDP_613 := [[10.82, 36.39, 5.21, 0, 48.4, 105.12], [9E9, 9E9, 9E9, 9E9, 9E9, 9E9]];
	VAR jointtarget CDP_614 := [[10.8, 36.38, 5.22, 0, 48.4, 104.44], [9E9, 9E9, 9E9, 9E9, 9E9, 9E9]];
	VAR jointtarget CDP_615 := [[10.79, 36.38, 5.23, 0, 48.39, 103.77], [9E9, 9E9, 9E9, 9E9, 9E9, 9E9]];
	VAR jointtarget CDP_616 := [[10.77, 36.37, 5.24, 0, 48.39, 103.09], [9E9, 9E9, 9E9, 9E9, 9E9, 9E9]];
	VAR jointtarget CDP_617 := [[10.75, 36.37, 5.24, 0, 48.39, 102.41], [9E9, 9E9, 9E9, 9E9, 9E9, 9E9]];
	VAR jointtarget CDP_618 := [[10.74, 36.37, 5.25, 0, 48.38, 101.73], [9E9, 9E9, 9E9, 9E9, 9E9, 9E9]];
	VAR jointtarget CDP_619 := [[10.72, 36.36, 5.26, 0, 48.38, 101.05], [9E9, 9E9, 9E9, 9E9, 9E9, 9E9]];
	VAR jointtarget CDP_620 := [[9.64, 36.15, 5.62, 0, 48.23, 99.64], [9E9, 9E9, 9E9, 9E9, 9E9, 9E9]];
	VAR jointtarget CDP_621 := [[8.56, 35.96, 5.94, 0, 48.1, 98.56], [9E9, 9E9, 9E9, 9E9, 9E9, 9E9]];
	VAR jointtarget CDP_622 := [[7.47, 35.8, 6.22, 0, 47.98, 97.47], [9E9, 9E9, 9E9, 9E9, 9E9, 9E9]];
	VAR jointtarget CDP_623 := [[6.38, 35.66, 6.47, 0, 47.87, 96.38], [9E9, 9E9, 9E9, 9E9, 9E9, 9E9]];
	VAR jointtarget CDP_624 := [[5.28, 35.54, 6.68, 0, 47.79, 95.28], [9E9, 9E9, 9E9, 9E9, 9E9, 9E9]];
	VAR jointtarget CDP_625 := [[4.17, 35.44, 6.84, 0, 47.72, 94.17], [9E9, 9E9, 9E9, 9E9, 9E9, 9E9]];
	VAR jointtarget CDP_626 := [[3.07, 35.36, 6.97, 0, 47.67, 93.07], [9E9, 9E9, 9E9, 9E9, 9E9, 9E9]];
	VAR jointtarget CDP_627 := [[1.96, 35.31, 7.06, 0, 47.63, 91.96], [9E9, 9E9, 9E9, 9E9, 9E9, 9E9]];
	VAR jointtarget CDP_628 := [[0.85, 35.28, 7.11, 0, 47.61, 90.85], [9E9, 9E9, 9E9, 9E9, 9E9, 9E9]];
	VAR jointtarget CDP_629 := [[-0.26, 35.28, 7.12, 0, 47.61, 89.74], [9E9, 9E9, 9E9, 9E9, 9E9, 9E9]];
	VAR jointtarget CDP_630 := [[-1.37, 35.29, 7.09, 0, 47.62, 88.63], [9E9, 9E9, 9E9, 9E9, 9E9, 9E9]];
	VAR jointtarget CDP_631 := [[-2.48, 35.33, 7.02, 0, 47.65, 87.52], [9E9, 9E9, 9E9, 9E9, 9E9, 9E9]];
	VAR jointtarget CDP_632 := [[-3.59, 35.4, 6.91, 0, 47.69, 86.41], [9E9, 9E9, 9E9, 9E9, 9E9, 9E9]];
	VAR jointtarget CDP_633 := [[-4.7, 35.48, 6.77, 0, 47.75, 85.3], [9E9, 9E9, 9E9, 9E9, 9E9, 9E9]];
	VAR jointtarget CDP_634 := [[-5.8, 35.59, 6.58, 0, 47.83, 84.2], [9E9, 9E9, 9E9, 9E9, 9E9, 9E9]];
	VAR jointtarget CDP_635 := [[-6.9, 35.72, 6.36, 0, 47.92, 83.1], [9E9, 9E9, 9E9, 9E9, 9E9, 9E9]];
	VAR jointtarget CDP_636 := [[-7.99, 35.87, 6.09, 0, 48.03, 82.01], [9E9, 9E9, 9E9, 9E9, 9E9, 9E9]];
	VAR jointtarget CDP_637 := [[-9.08, 36.05, 5.79, 0, 48.16, 80.92], [9E9, 9E9, 9E9, 9E9, 9E9, 9E9]];
	VAR jointtarget CDP_638 := [[-10.16, 36.25, 5.45, 0, 48.3, 79.84], [9E9, 9E9, 9E9, 9E9, 9E9, 9E9]];
	VAR jointtarget CDP_639 := [[-11.23, 36.47, 5.07, 0, 48.46, 78.77], [9E9, 9E9, 9E9, 9E9, 9E9, 9E9]];
	VAR jointtarget CDP_640 := [[-11.28, 36.48, 5.05, 0, 48.47, 79.81], [9E9, 9E9, 9E9, 9E9, 9E9, 9E9]];
	VAR jointtarget CDP_641 := [[-11.34, 36.49, 5.04, 0, 48.47, 81.95], [9E9, 9E9, 9E9, 9E9, 9E9, 9E9]];
	VAR jointtarget CDP_642 := [[-11.39, 36.5, 5.03, 0, 48.48, 84.09], [9E9, 9E9, 9E9, 9E9, 9E9, 9E9]];
	VAR jointtarget CDP_643 := [[-11.45, 36.5, 5.02, 0, 48.48, 86.23], [9E9, 9E9, 9E9, 9E9, 9E9, 9E9]];
	VAR jointtarget CDP_644 := [[-11.5, 36.5, 5.02, 0, 48.48, 88.37], [9E9, 9E9, 9E9, 9E9, 9E9, 9E9]];
	VAR jointtarget CDP_645 := [[-11.56, 36.5, 5.02, 0, 48.48, 90.51], [9E9, 9E9, 9E9, 9E9, 9E9, 9E9]];
	VAR jointtarget CDP_646 := [[-11.61, 36.5, 5.02, 0, 48.48, 92.65], [9E9, 9E9, 9E9, 9E9, 9E9, 9E9]];
	VAR jointtarget CDP_647 := [[-11.67, 36.49, 5.03, 0, 48.47, 94.78], [9E9, 9E9, 9E9, 9E9, 9E9, 9E9]];
	VAR jointtarget CDP_648 := [[-11.72, 36.49, 5.04, 0, 48.47, 96.92], [9E9, 9E9, 9E9, 9E9, 9E9, 9E9]];
	VAR jointtarget CDP_649 := [[-11.78, 36.48, 5.06, 0, 48.46, 99.06], [9E9, 9E9, 9E9, 9E9, 9E9, 9E9]];
	VAR jointtarget CDP_650 := [[-11.83, 36.47, 5.08, 0, 48.45, 101.2], [9E9, 9E9, 9E9, 9E9, 9E9, 9E9]];
	VAR jointtarget CDP_651 := [[-11.89, 36.45, 5.1, 0, 48.44, 103.34], [9E9, 9E9, 9E9, 9E9, 9E9, 9E9]];
	VAR jointtarget CDP_652 := [[-11.94, 36.44, 5.13, 0, 48.43, 105.48], [9E9, 9E9, 9E9, 9E9, 9E9, 9E9]];
	VAR jointtarget CDP_653 := [[-11.99, 36.42, 5.16, 0, 48.42, 107.63], [9E9, 9E9, 9E9, 9E9, 9E9, 9E9]];
	VAR jointtarget CDP_654 := [[-12.04, 36.4, 5.2, 0, 48.4, 109.77], [9E9, 9E9, 9E9, 9E9, 9E9, 9E9]];
	VAR jointtarget CDP_655 := [[-12.09, 36.37, 5.24, 0, 48.39, 111.91], [9E9, 9E9, 9E9, 9E9, 9E9, 9E9]];
	VAR jointtarget CDP_656 := [[-12.15, 36.35, 5.28, 0, 48.37, 114.05], [9E9, 9E9, 9E9, 9E9, 9E9, 9E9]];
	VAR jointtarget CDP_657 := [[-12.19, 36.32, 5.33, 0, 48.35, 116.2], [9E9, 9E9, 9E9, 9E9, 9E9, 9E9]];
	VAR jointtarget CDP_658 := [[-12.24, 36.29, 5.38, 0, 48.33, 118.34], [9E9, 9E9, 9E9, 9E9, 9E9, 9E9]];
	VAR jointtarget CDP_659 := [[-12.29, 36.26, 5.43, 0, 48.31, 120.49], [9E9, 9E9, 9E9, 9E9, 9E9, 9E9]];
	VAR jointtarget CDP_660 := [[-12.32, 36.24, 5.46, 0, 48.3, 121.56], [9E9, 9E9, 9E9, 9E9, 9E9, 9E9]];
	VAR jointtarget CDP_661 := [[-12.35, 36.22, 5.49, 0, 48.28, 121.53], [9E9, 9E9, 9E9, 9E9, 9E9, 9E9]];
	VAR jointtarget CDP_662 := [[-12.38, 36.21, 5.53, 0, 48.27, 121.5], [9E9, 9E9, 9E9, 9E9, 9E9, 9E9]];
	VAR jointtarget CDP_663 := [[-12.41, 36.19, 5.56, 0, 48.25, 121.47], [9E9, 9E9, 9E9, 9E9, 9E9, 9E9]];
	VAR jointtarget CDP_664 := [[-12.43, 36.17, 5.59, 0, 48.24, 121.44], [9E9, 9E9, 9E9, 9E9, 9E9, 9E9]];
	VAR jointtarget CDP_665 := [[-12.46, 36.15, 5.62, 0, 48.23, 121.41], [9E9, 9E9, 9E9, 9E9, 9E9, 9E9]];
	VAR jointtarget CDP_666 := [[-12.49, 36.13, 5.66, 0, 48.21, 121.39], [9E9, 9E9, 9E9, 9E9, 9E9, 9E9]];
	VAR jointtarget CDP_667 := [[-12.52, 36.11, 5.69, 0, 48.2, 121.36], [9E9, 9E9, 9E9, 9E9, 9E9, 9E9]];
	VAR jointtarget CDP_668 := [[-12.55, 36.09, 5.72, 0, 48.19, 121.33], [9E9, 9E9, 9E9, 9E9, 9E9, 9E9]];
	VAR jointtarget CDP_669 := [[-12.58, 36.07, 5.75, 0, 48.17, 121.3], [9E9, 9E9, 9E9, 9E9, 9E9, 9E9]];
	VAR jointtarget CDP_670 := [[-12.61, 36.05, 5.79, 0, 48.16, 121.27], [9E9, 9E9, 9E9, 9E9, 9E9, 9E9]];
	VAR jointtarget CDP_671 := [[-12.63, 36.04, 5.82, 0, 48.15, 121.24], [9E9, 9E9, 9E9, 9E9, 9E9, 9E9]];
	VAR jointtarget CDP_672 := [[-12.66, 36.02, 5.85, 0, 48.13, 121.21], [9E9, 9E9, 9E9, 9E9, 9E9, 9E9]];
	VAR jointtarget CDP_673 := [[-12.69, 36, 5.88, 0, 48.12, 121.18], [9E9, 9E9, 9E9, 9E9, 9E9, 9E9]];
	VAR jointtarget CDP_674 := [[-12.72, 35.98, 5.92, 0, 48.11, 121.16], [9E9, 9E9, 9E9, 9E9, 9E9, 9E9]];
	VAR jointtarget CDP_675 := [[-12.75, 35.96, 5.95, 0, 48.09, 121.13], [9E9, 9E9, 9E9, 9E9, 9E9, 9E9]];
	VAR jointtarget CDP_676 := [[-12.78, 35.94, 5.98, 0, 48.08, 121.1], [9E9, 9E9, 9E9, 9E9, 9E9, 9E9]];
	VAR jointtarget CDP_677 := [[-12.81, 35.92, 6.01, 0, 48.06, 121.07], [9E9, 9E9, 9E9, 9E9, 9E9, 9E9]];
	VAR jointtarget CDP_678 := [[-12.84, 35.9, 6.04, 0, 48.05, 121.04], [9E9, 9E9, 9E9, 9E9, 9E9, 9E9]];
	VAR jointtarget CDP_679 := [[-12.86, 35.88, 6.08, 0, 48.04, 121.01], [9E9, 9E9, 9E9, 9E9, 9E9, 9E9]];
	VAR jointtarget CDP_680 := [[-13.02, 35.81, 6.2, 0, 47.99, 114.17], [9E9, 9E9, 9E9, 9E9, 9E9, 9E9]];
	VAR jointtarget CDP_681 := [[-13.18, 35.78, 6.26, 0, 47.96, 100.62], [9E9, 9E9, 9E9, 9E9, 9E9, 9E9]];
	VAR jointtarget CDP_682 := [[-13.34, 35.79, 6.24, 0, 47.97, 87.07], [9E9, 9E9, 9E9, 9E9, 9E9, 9E9]];
	VAR jointtarget CDP_683 := [[-13.5, 35.84, 6.16, 0, 48, 73.52], [9E9, 9E9, 9E9, 9E9, 9E9, 9E9]];
	VAR jointtarget CDP_684 := [[-13.64, 35.93, 6.01, 0, 48.07, 59.99], [9E9, 9E9, 9E9, 9E9, 9E9, 9E9]];
	VAR jointtarget CDP_685 := [[-13.76, 36.05, 5.8, 0, 48.16, 46.48], [9E9, 9E9, 9E9, 9E9, 9E9, 9E9]];
	VAR jointtarget CDP_686 := [[-13.85, 36.2, 5.54, 0, 48.26, 33.01], [9E9, 9E9, 9E9, 9E9, 9E9, 9E9]];
	VAR jointtarget CDP_687 := [[-13.91, 36.37, 5.25, 0, 48.38, 19.56], [9E9, 9E9, 9E9, 9E9, 9E9, 9E9]];
	VAR jointtarget CDP_688 := [[-13.92, 36.54, 4.95, 0, 48.51, 6.16], [9E9, 9E9, 9E9, 9E9, 9E9, 9E9]];
	VAR jointtarget CDP_689 := [[-13.9, 36.72, 4.64, 0, 48.64, -7.21], [9E9, 9E9, 9E9, 9E9, 9E9, 9E9]];
	VAR jointtarget CDP_690 := [[-13.85, 36.89, 4.35, 0, 48.76, -20.54], [9E9, 9E9, 9E9, 9E9, 9E9, 9E9]];
	VAR jointtarget CDP_691 := [[-13.76, 37.04, 4.09, 0, 48.87, -33.84], [9E9, 9E9, 9E9, 9E9, 9E9, 9E9]];
	VAR jointtarget CDP_692 := [[-13.64, 37.16, 3.88, 0, 48.96, -47.11], [9E9, 9E9, 9E9, 9E9, 9E9, 9E9]];
	VAR jointtarget CDP_693 := [[-13.5, 37.25, 3.73, 0, 49.02, -60.35], [9E9, 9E9, 9E9, 9E9, 9E9, 9E9]];
	VAR jointtarget CDP_694 := [[-13.34, 37.3, 3.64, 0, 49.06, -73.59], [9E9, 9E9, 9E9, 9E9, 9E9, 9E9]];
	VAR jointtarget CDP_695 := [[-13.18, 37.31, 3.63, 0, 49.07, -86.81], [9E9, 9E9, 9E9, 9E9, 9E9, 9E9]];
	VAR jointtarget CDP_696 := [[-13.02, 37.28, 3.68, 0, 49.04, -100.04], [9E9, 9E9, 9E9, 9E9, 9E9, 9E9]];
	VAR jointtarget CDP_697 := [[-12.88, 37.21, 3.8, 0, 48.99, -113.28], [9E9, 9E9, 9E9, 9E9, 9E9, 9E9]];
	VAR jointtarget CDP_698 := [[-12.75, 37.1, 3.99, 0, 48.91, -126.54], [9E9, 9E9, 9E9, 9E9, 9E9, 9E9]];
	VAR jointtarget CDP_699 := [[-12.64, 36.96, 4.22, 0, 48.81, -139.82], [9E9, 9E9, 9E9, 9E9, 9E9, 9E9]];
	VAR jointtarget CDP_700 := [[-12.62, 36.92, 4.3, 0, 48.78, -146.49], [9E9, 9E9, 9E9, 9E9, 9E9, 9E9]];
	VAR jointtarget CDP_701 := [[-12.59, 36.88, 4.37, 0, 48.75, -146.47], [9E9, 9E9, 9E9, 9E9, 9E9, 9E9]];
	VAR jointtarget CDP_702 := [[-12.57, 36.84, 4.44, 0, 48.72, -146.44], [9E9, 9E9, 9E9, 9E9, 9E9, 9E9]];
	VAR jointtarget CDP_703 := [[-12.54, 36.8, 4.51, 0, 48.69, -146.42], [9E9, 9E9, 9E9, 9E9, 9E9, 9E9]];
	VAR jointtarget CDP_704 := [[-12.52, 36.76, 4.58, 0, 48.66, -146.4], [9E9, 9E9, 9E9, 9E9, 9E9, 9E9]];
	VAR jointtarget CDP_705 := [[-12.49, 36.72, 4.65, 0, 48.63, -146.37], [9E9, 9E9, 9E9, 9E9, 9E9, 9E9]];
	VAR jointtarget CDP_706 := [[-12.47, 36.67, 4.72, 0, 48.6, -146.35], [9E9, 9E9, 9E9, 9E9, 9E9, 9E9]];
	VAR jointtarget CDP_707 := [[-12.44, 36.63, 4.79, 0, 48.58, -146.32], [9E9, 9E9, 9E9, 9E9, 9E9, 9E9]];
	VAR jointtarget CDP_708 := [[-12.42, 36.59, 4.86, 0, 48.55, -146.3], [9E9, 9E9, 9E9, 9E9, 9E9, 9E9]];
	VAR jointtarget CDP_709 := [[-12.39, 36.55, 4.93, 0, 48.52, -146.27], [9E9, 9E9, 9E9, 9E9, 9E9, 9E9]];
	VAR jointtarget CDP_710 := [[-12.37, 36.51, 5, 0, 48.49, -146.25], [9E9, 9E9, 9E9, 9E9, 9E9, 9E9]];
	VAR jointtarget CDP_711 := [[-12.34, 36.47, 5.07, 0, 48.46, -146.22], [9E9, 9E9, 9E9, 9E9, 9E9, 9E9]];
	VAR jointtarget CDP_712 := [[-12.32, 36.43, 5.14, 0, 48.43, -146.2], [9E9, 9E9, 9E9, 9E9, 9E9, 9E9]];
	VAR jointtarget CDP_713 := [[-12.29, 36.39, 5.21, 0, 48.4, -146.17], [9E9, 9E9, 9E9, 9E9, 9E9, 9E9]];
	VAR jointtarget CDP_714 := [[-12.27, 36.35, 5.28, 0, 48.37, -146.15], [9E9, 9E9, 9E9, 9E9, 9E9, 9E9]];
	VAR jointtarget CDP_715 := [[-12.24, 36.31, 5.35, 0, 48.34, -146.12], [9E9, 9E9, 9E9, 9E9, 9E9, 9E9]];
	VAR jointtarget CDP_716 := [[-12.22, 36.27, 5.42, 0, 48.31, -146.1], [9E9, 9E9, 9E9, 9E9, 9E9, 9E9]];
	VAR jointtarget CDP_717 := [[-12.19, 36.22, 5.49, 0, 48.28, -146.07], [9E9, 9E9, 9E9, 9E9, 9E9, 9E9]];
	VAR jointtarget CDP_718 := [[-12.17, 36.18, 5.56, 0, 48.25, -146.05], [9E9, 9E9, 9E9, 9E9, 9E9, 9E9]];
	VAR jointtarget CDP_719 := [[-12.14, 36.14, 5.63, 0, 48.22, -146.02], [9E9, 9E9, 9E9, 9E9, 9E9, 9E9]];
	VAR jointtarget CDP_720 := [[-12.14, 36.13, 5.66, 0, 48.21, -145.46], [9E9, 9E9, 9E9, 9E9, 9E9, 9E9]];
	VAR jointtarget CDP_721 := [[-12.13, 36.12, 5.68, 0, 48.21, -144.35], [9E9, 9E9, 9E9, 9E9, 9E9, 9E9]];
	VAR jointtarget CDP_722 := [[-12.12, 36.11, 5.7, 0, 48.2, -143.24], [9E9, 9E9, 9E9, 9E9, 9E9, 9E9]];
	VAR jointtarget CDP_723 := [[-12.11, 36.09, 5.72, 0, 48.19, -142.13], [9E9, 9E9, 9E9, 9E9, 9E9, 9E9]];
	VAR jointtarget CDP_724 := [[-12.1, 36.08, 5.74, 0, 48.18, -141.01], [9E9, 9E9, 9E9, 9E9, 9E9, 9E9]];
	VAR jointtarget CDP_725 := [[-12.09, 36.07, 5.76, 0, 48.17, -139.9], [9E9, 9E9, 9E9, 9E9, 9E9, 9E9]];
	VAR jointtarget CDP_726 := [[-12.08, 36.06, 5.78, 0, 48.16, -138.79], [9E9, 9E9, 9E9, 9E9, 9E9, 9E9]];
	VAR jointtarget CDP_727 := [[-12.07, 36.05, 5.8, 0, 48.16, -137.68], [9E9, 9E9, 9E9, 9E9, 9E9, 9E9]];
	VAR jointtarget CDP_728 := [[-12.06, 36.04, 5.82, 0, 48.15, -136.56], [9E9, 9E9, 9E9, 9E9, 9E9, 9E9]];
	VAR jointtarget CDP_729 := [[-12.05, 36.02, 5.83, 0, 48.14, -135.45], [9E9, 9E9, 9E9, 9E9, 9E9, 9E9]];
	VAR jointtarget CDP_730 := [[-12.04, 36.01, 5.85, 0, 48.13, -134.34], [9E9, 9E9, 9E9, 9E9, 9E9, 9E9]];
	VAR jointtarget CDP_731 := [[-12.03, 36, 5.87, 0, 48.13, -133.22], [9E9, 9E9, 9E9, 9E9, 9E9, 9E9]];
	VAR jointtarget CDP_732 := [[-12.02, 35.99, 5.89, 0, 48.12, -132.11], [9E9, 9E9, 9E9, 9E9, 9E9, 9E9]];
	VAR jointtarget CDP_733 := [[-12.01, 35.98, 5.91, 0, 48.11, -130.99], [9E9, 9E9, 9E9, 9E9, 9E9, 9E9]];
	VAR jointtarget CDP_734 := [[-12, 35.97, 5.92, 0, 48.11, -129.88], [9E9, 9E9, 9E9, 9E9, 9E9, 9E9]];
	VAR jointtarget CDP_735 := [[-11.99, 35.96, 5.94, 0, 48.1, -128.76], [9E9, 9E9, 9E9, 9E9, 9E9, 9E9]];
	VAR jointtarget CDP_736 := [[-11.98, 35.95, 5.95, 0, 48.09, -127.65], [9E9, 9E9, 9E9, 9E9, 9E9, 9E9]];
	VAR jointtarget CDP_737 := [[-11.97, 35.94, 5.97, 0, 48.09, -126.53], [9E9, 9E9, 9E9, 9E9, 9E9, 9E9]];
	VAR jointtarget CDP_738 := [[-11.96, 35.93, 5.98, 0, 48.08, -125.42], [9E9, 9E9, 9E9, 9E9, 9E9, 9E9]];
	VAR jointtarget CDP_739 := [[-11.95, 35.92, 6, 0, 48.08, -124.3], [9E9, 9E9, 9E9, 9E9, 9E9, 9E9]];
	VAR jointtarget CDP_740 := [[-11.94, 35.92, 6.01, 0, 48.07, -123.74], [9E9, 9E9, 9E9, 9E9, 9E9, 9E9]];
	VAR jointtarget CDP_741 := [[-11.93, 35.91, 6.02, 0, 48.07, -123.73], [9E9, 9E9, 9E9, 9E9, 9E9, 9E9]];
	VAR jointtarget CDP_742 := [[-11.92, 35.9, 6.04, 0, 48.06, -123.72], [9E9, 9E9, 9E9, 9E9, 9E9, 9E9]];
	VAR jointtarget CDP_743 := [[-11.9, 35.89, 6.05, 0, 48.06, -123.71], [9E9, 9E9, 9E9, 9E9, 9E9, 9E9]];
	VAR jointtarget CDP_744 := [[-11.89, 35.89, 6.06, 0, 48.05, -123.7], [9E9, 9E9, 9E9, 9E9, 9E9, 9E9]];
	VAR jointtarget CDP_745 := [[-11.88, 35.88, 6.08, 0, 48.05, -123.69], [9E9, 9E9, 9E9, 9E9, 9E9, 9E9]];
	VAR jointtarget CDP_746 := [[-11.87, 35.87, 6.09, 0, 48.04, -123.68], [9E9, 9E9, 9E9, 9E9, 9E9, 9E9]];
	VAR jointtarget CDP_747 := [[-11.86, 35.86, 6.1, 0, 48.04, -123.66], [9E9, 9E9, 9E9, 9E9, 9E9, 9E9]];
	VAR jointtarget CDP_748 := [[-11.85, 35.85, 6.11, 0, 48.03, -123.65], [9E9, 9E9, 9E9, 9E9, 9E9, 9E9]];
	VAR jointtarget CDP_749 := [[-11.84, 35.85, 6.13, 0, 48.03, -123.64], [9E9, 9E9, 9E9, 9E9, 9E9, 9E9]];
	VAR jointtarget CDP_750 := [[-11.83, 35.84, 6.14, 0, 48.02, -123.63], [9E9, 9E9, 9E9, 9E9, 9E9, 9E9]];
	VAR jointtarget CDP_751 := [[-11.82, 35.83, 6.15, 0, 48.02, -123.62], [9E9, 9E9, 9E9, 9E9, 9E9, 9E9]];
	VAR jointtarget CDP_752 := [[-11.81, 35.82, 6.16, 0, 48.01, -123.61], [9E9, 9E9, 9E9, 9E9, 9E9, 9E9]];
	VAR jointtarget CDP_753 := [[-11.8, 35.81, 6.18, 0, 48.01, -123.6], [9E9, 9E9, 9E9, 9E9, 9E9, 9E9]];
	VAR jointtarget CDP_754 := [[-11.79, 35.81, 6.19, 0, 48, -123.59], [9E9, 9E9, 9E9, 9E9, 9E9, 9E9]];
	VAR jointtarget CDP_755 := [[-11.78, 35.8, 6.2, 0, 48, -123.58], [9E9, 9E9, 9E9, 9E9, 9E9, 9E9]];
	VAR jointtarget CDP_756 := [[-11.77, 35.79, 6.22, 0, 47.99, -123.57], [9E9, 9E9, 9E9, 9E9, 9E9, 9E9]];
	VAR jointtarget CDP_757 := [[-11.76, 35.78, 6.23, 0, 47.99, -123.56], [9E9, 9E9, 9E9, 9E9, 9E9, 9E9]];
	VAR jointtarget CDP_758 := [[-11.75, 35.78, 6.24, 0, 47.98, -123.55], [9E9, 9E9, 9E9, 9E9, 9E9, 9E9]];
	VAR jointtarget CDP_759 := [[-11.74, 35.77, 6.25, 0, 47.98, -123.54], [9E9, 9E9, 9E9, 9E9, 9E9, 9E9]];
	VAR jointtarget CDP_760 := [[-10.65, 35.54, 6.65, 0, 47.81, -100.65], [9E9, 9E9, 9E9, 9E9, 9E9, 9E9]];
	VAR jointtarget CDP_761 := [[-9.55, 35.33, 7.01, 0, 47.67, -99.55], [9E9, 9E9, 9E9, 9E9, 9E9, 9E9]];
	VAR jointtarget CDP_762 := [[-8.44, 35.14, 7.33, 0, 47.53, -98.44], [9E9, 9E9, 9E9, 9E9, 9E9, 9E9]];
	VAR jointtarget CDP_763 := [[-7.33, 34.98, 7.6, 0, 47.42, -97.33], [9E9, 9E9, 9E9, 9E9, 9E9, 9E9]];
	VAR jointtarget CDP_764 := [[-6.21, 34.84, 7.84, 0, 47.32, -96.21], [9E9, 9E9, 9E9, 9E9, 9E9, 9E9]];
	VAR jointtarget CDP_765 := [[-5.09, 34.72, 8.04, 0, 47.24, -95.09], [9E9, 9E9, 9E9, 9E9, 9E9, 9E9]];
	VAR jointtarget CDP_766 := [[-3.96, 34.63, 8.2, 0, 47.17, -93.96], [9E9, 9E9, 9E9, 9E9, 9E9, 9E9]];
	VAR jointtarget CDP_767 := [[-2.83, 34.56, 8.32, 0, 47.12, -92.83], [9E9, 9E9, 9E9, 9E9, 9E9, 9E9]];
	VAR jointtarget CDP_768 := [[-1.7, 34.51, 8.4, 0, 47.09, -91.7], [9E9, 9E9, 9E9, 9E9, 9E9, 9E9]];
	VAR jointtarget CDP_769 := [[-0.56, 34.49, 8.44, 0, 47.07, -90.56], [9E9, 9E9, 9E9, 9E9, 9E9, 9E9]];
	VAR jointtarget CDP_770 := [[0.57, 34.49, 8.44, 0, 47.07, -89.43], [9E9, 9E9, 9E9, 9E9, 9E9, 9E9]];
	VAR jointtarget CDP_771 := [[1.7, 34.51, 8.4, 0, 47.09, -88.3], [9E9, 9E9, 9E9, 9E9, 9E9, 9E9]];
	VAR jointtarget CDP_772 := [[2.84, 34.56, 8.32, 0, 47.12, -87.16], [9E9, 9E9, 9E9, 9E9, 9E9, 9E9]];
	VAR jointtarget CDP_773 := [[3.97, 34.63, 8.2, 0, 47.17, -86.03], [9E9, 9E9, 9E9, 9E9, 9E9, 9E9]];
	VAR jointtarget CDP_774 := [[5.09, 34.72, 8.04, 0, 47.24, -84.91], [9E9, 9E9, 9E9, 9E9, 9E9, 9E9]];
	VAR jointtarget CDP_775 := [[6.22, 34.84, 7.84, 0, 47.32, -83.78], [9E9, 9E9, 9E9, 9E9, 9E9, 9E9]];
	VAR jointtarget CDP_776 := [[7.34, 34.98, 7.6, 0, 47.42, -82.66], [9E9, 9E9, 9E9, 9E9, 9E9, 9E9]];
	VAR jointtarget CDP_777 := [[8.45, 35.14, 7.32, 0, 47.53, -81.55], [9E9, 9E9, 9E9, 9E9, 9E9, 9E9]];
	VAR jointtarget CDP_778 := [[9.56, 35.33, 7.01, 0, 47.67, -80.44], [9E9, 9E9, 9E9, 9E9, 9E9, 9E9]];
	VAR jointtarget CDP_779 := [[10.65, 35.54, 6.65, 0, 47.82, -79.35], [9E9, 9E9, 9E9, 9E9, 9E9, 9E9]];
	VAR jointtarget CDP_780 := [[10.71, 35.55, 6.63, 0, 47.82, -78.19], [9E9, 9E9, 9E9, 9E9, 9E9, 9E9]];
	VAR jointtarget CDP_781 := [[10.76, 35.56, 6.6, 0, 47.83, -75.95], [9E9, 9E9, 9E9, 9E9, 9E9, 9E9]];
	VAR jointtarget CDP_782 := [[10.82, 35.58, 6.57, 0, 47.85, -73.7], [9E9, 9E9, 9E9, 9E9, 9E9, 9E9]];
	VAR jointtarget CDP_783 := [[10.87, 35.6, 6.54, 0, 47.86, -71.45], [9E9, 9E9, 9E9, 9E9, 9E9, 9E9]];
	VAR jointtarget CDP_784 := [[10.92, 35.62, 6.5, 0, 47.87, -69.2], [9E9, 9E9, 9E9, 9E9, 9E9, 9E9]];
	VAR jointtarget CDP_785 := [[10.97, 35.64, 6.46, 0, 47.89, -66.96], [9E9, 9E9, 9E9, 9E9, 9E9, 9E9]];
	VAR jointtarget CDP_786 := [[11.03, 35.67, 6.42, 0, 47.91, -64.72], [9E9, 9E9, 9E9, 9E9, 9E9, 9E9]];
	VAR jointtarget CDP_787 := [[11.07, 35.7, 6.37, 0, 47.93, -62.47], [9E9, 9E9, 9E9, 9E9, 9E9, 9E9]];
	VAR jointtarget CDP_788 := [[11.12, 35.73, 6.32, 0, 47.95, -60.23], [9E9, 9E9, 9E9, 9E9, 9E9, 9E9]];
	VAR jointtarget CDP_789 := [[11.17, 35.76, 6.27, 0, 47.97, -57.99], [9E9, 9E9, 9E9, 9E9, 9E9, 9E9]];
	VAR jointtarget CDP_790 := [[11.22, 35.79, 6.21, 0, 48, -55.75], [9E9, 9E9, 9E9, 9E9, 9E9, 9E9]];
	VAR jointtarget CDP_791 := [[11.26, 35.83, 6.15, 0, 48.02, -53.51], [9E9, 9E9, 9E9, 9E9, 9E9, 9E9]];
	VAR jointtarget CDP_792 := [[11.3, 35.87, 6.08, 0, 48.05, -51.27], [9E9, 9E9, 9E9, 9E9, 9E9, 9E9]];
	VAR jointtarget CDP_793 := [[11.35, 35.91, 6.02, 0, 48.08, -49.04], [9E9, 9E9, 9E9, 9E9, 9E9, 9E9]];
	VAR jointtarget CDP_794 := [[11.39, 35.95, 5.95, 0, 48.11, -46.8], [9E9, 9E9, 9E9, 9E9, 9E9, 9E9]];
	VAR jointtarget CDP_795 := [[11.43, 35.99, 5.87, 0, 48.14, -44.57], [9E9, 9E9, 9E9, 9E9, 9E9, 9E9]];
	VAR jointtarget CDP_796 := [[11.46, 36.03, 5.8, 0, 48.17, -42.34], [9E9, 9E9, 9E9, 9E9, 9E9, 9E9]];
	VAR jointtarget CDP_797 := [[11.5, 36.08, 5.72, 0, 48.2, -40.11], [9E9, 9E9, 9E9, 9E9, 9E9, 9E9]];
	VAR jointtarget CDP_798 := [[11.53, 36.13, 5.63, 0, 48.24, -37.88], [9E9, 9E9, 9E9, 9E9, 9E9, 9E9]];
	VAR jointtarget CDP_799 := [[11.57, 36.18, 5.55, 0, 48.27, -35.65], [9E9, 9E9, 9E9, 9E9, 9E9, 9E9]];
	VAR jointtarget CDP_800 := [[11.59, 36.21, 5.5, 0, 48.29, -34.54], [9E9, 9E9, 9E9, 9E9, 9E9, 9E9]];
	VAR jointtarget CDP_801 := [[11.6, 36.24, 5.45, 0, 48.32, -34.52], [9E9, 9E9, 9E9, 9E9, 9E9, 9E9]];
	VAR jointtarget CDP_802 := [[11.62, 36.27, 5.4, 0, 48.34, -34.5], [9E9, 9E9, 9E9, 9E9, 9E9, 9E9]];
	VAR jointtarget CDP_803 := [[11.64, 36.3, 5.34, 0, 48.36, -34.48], [9E9, 9E9, 9E9, 9E9, 9E9, 9E9]];
	VAR jointtarget CDP_804 := [[11.66, 36.33, 5.29, 0, 48.38, -34.46], [9E9, 9E9, 9E9, 9E9, 9E9, 9E9]];
	VAR jointtarget CDP_805 := [[11.68, 36.36, 5.24, 0, 48.4, -34.44], [9E9, 9E9, 9E9, 9E9, 9E9, 9E9]];
	VAR jointtarget CDP_806 := [[11.7, 36.39, 5.19, 0, 48.42, -34.42], [9E9, 9E9, 9E9, 9E9, 9E9, 9E9]];
	VAR jointtarget CDP_807 := [[11.72, 36.42, 5.14, 0, 48.44, -34.41], [9E9, 9E9, 9E9, 9E9, 9E9, 9E9]];
	VAR jointtarget CDP_808 := [[11.74, 36.45, 5.09, 0, 48.47, -34.39], [9E9, 9E9, 9E9, 9E9, 9E9, 9E9]];
	VAR jointtarget CDP_809 := [[11.76, 36.48, 5.03, 0, 48.49, -34.37], [9E9, 9E9, 9E9, 9E9, 9E9, 9E9]];
	VAR jointtarget CDP_810 := [[11.77, 36.51, 4.98, 0, 48.51, -34.35], [9E9, 9E9, 9E9, 9E9, 9E9, 9E9]];
	VAR jointtarget CDP_811 := [[11.79, 36.54, 4.93, 0, 48.53, -34.33], [9E9, 9E9, 9E9, 9E9, 9E9, 9E9]];
	VAR jointtarget CDP_812 := [[11.81, 36.57, 4.88, 0, 48.55, -34.31], [9E9, 9E9, 9E9, 9E9, 9E9, 9E9]];
	VAR jointtarget CDP_813 := [[11.83, 36.6, 4.83, 0, 48.58, -34.29], [9E9, 9E9, 9E9, 9E9, 9E9, 9E9]];
	VAR jointtarget CDP_814 := [[11.85, 36.63, 4.77, 0, 48.6, -34.27], [9E9, 9E9, 9E9, 9E9, 9E9, 9E9]];
	VAR jointtarget CDP_815 := [[11.87, 36.66, 4.72, 0, 48.62, -34.26], [9E9, 9E9, 9E9, 9E9, 9E9, 9E9]];
	VAR jointtarget CDP_816 := [[11.89, 36.69, 4.67, 0, 48.64, -34.24], [9E9, 9E9, 9E9, 9E9, 9E9, 9E9]];
	VAR jointtarget CDP_817 := [[11.91, 36.72, 4.62, 0, 48.66, -34.22], [9E9, 9E9, 9E9, 9E9, 9E9, 9E9]];
	VAR jointtarget CDP_818 := [[11.92, 36.75, 4.57, 0, 48.68, -34.2], [9E9, 9E9, 9E9, 9E9, 9E9, 9E9]];
	VAR jointtarget CDP_819 := [[11.94, 36.78, 4.51, 0, 48.71, -34.18], [9E9, 9E9, 9E9, 9E9, 9E9, 9E9]];
	VAR jointtarget CDP_820 := [[12.05, 36.92, 4.28, 0, 48.8, -40.77], [9E9, 9E9, 9E9, 9E9, 9E9, 9E9]];
	VAR jointtarget CDP_821 := [[12.18, 37.02, 4.1, 0, 48.88, -54.03], [9E9, 9E9, 9E9, 9E9, 9E9, 9E9]];
	VAR jointtarget CDP_822 := [[12.33, 37.09, 3.98, 0, 48.93, -67.26], [9E9, 9E9, 9E9, 9E9, 9E9, 9E9]];
	VAR jointtarget CDP_823 := [[12.49, 37.12, 3.93, 0, 48.95, -80.49], [9E9, 9E9, 9E9, 9E9, 9E9, 9E9]];
	VAR jointtarget CDP_824 := [[12.65, 37.11, 3.95, 0, 48.94, -93.72], [9E9, 9E9, 9E9, 9E9, 9E9, 9E9]];
	VAR jointtarget CDP_825 := [[12.8, 37.06, 4.04, 0, 48.91, -106.95], [9E9, 9E9, 9E9, 9E9, 9E9, 9E9]];
	VAR jointtarget CDP_826 := [[12.94, 36.96, 4.2, 0, 48.84, -120.2], [9E9, 9E9, 9E9, 9E9, 9E9, 9E9]];
	VAR jointtarget CDP_827 := [[13.06, 36.84, 4.41, 0, 48.75, -133.47], [9E9, 9E9, 9E9, 9E9, 9E9, 9E9]];
	VAR jointtarget CDP_828 := [[13.15, 36.69, 4.67, 0, 48.64, -146.77], [9E9, 9E9, 9E9, 9E9, 9E9, 9E9]];
	VAR jointtarget CDP_829 := [[13.2, 36.52, 4.96, 0, 48.52, -160.1], [9E9, 9E9, 9E9, 9E9, 9E9, 9E9]];
	VAR jointtarget CDP_830 := [[13.22, 36.35, 5.26, 0, 48.39, -173.47], [9E9, 9E9, 9E9, 9E9, 9E9, 9E9]];
	VAR jointtarget CDP_831 := [[13.2, 36.17, 5.57, 0, 48.27, -186.88], [9E9, 9E9, 9E9, 9E9, 9E9, 9E9]];
	VAR jointtarget CDP_832 := [[13.15, 36, 5.85, 0, 48.15, -200.32], [9E9, 9E9, 9E9, 9E9, 9E9, 9E9]];
	VAR jointtarget CDP_833 := [[13.06, 35.85, 6.11, 0, 48.04, -213.8], [9E9, 9E9, 9E9, 9E9, 9E9, 9E9]];
	VAR jointtarget CDP_834 := [[12.93, 35.73, 6.31, 0, 47.95, -227.31], [9E9, 9E9, 9E9, 9E9, 9E9, 9E9]];
	VAR jointtarget CDP_835 := [[12.79, 35.65, 6.46, 0, 47.89, -240.84], [9E9, 9E9, 9E9, 9E9, 9E9, 9E9]];
	VAR jointtarget CDP_836 := [[12.63, 35.6, 6.54, 0, 47.86, -254.39], [9E9, 9E9, 9E9, 9E9, 9E9, 9E9]];
	VAR jointtarget CDP_837 := [[12.47, 35.59, 6.55, 0, 47.85, -267.94], [9E9, 9E9, 9E9, 9E9, 9E9, 9E9]];
	VAR jointtarget CDP_838 := [[12.3, 35.63, 6.49, 0, 47.88, -281.49], [9E9, 9E9, 9E9, 9E9, 9E9, 9E9]];
	VAR jointtarget CDP_839 := [[12.15, 35.7, 6.37, 0, 47.93, -295.03], [9E9, 9E9, 9E9, 9E9, 9E9, 9E9]];
	VAR jointtarget CDP_840 := [[12.13, 35.72, 6.33, 0, 47.95, -301.75], [9E9, 9E9, 9E9, 9E9, 9E9, 9E9]];
	VAR jointtarget CDP_841 := [[12.1, 35.74, 6.3, 0, 47.96, -301.78], [9E9, 9E9, 9E9, 9E9, 9E9, 9E9]];
	VAR jointtarget CDP_842 := [[12.07, 35.76, 6.27, 0, 47.97, -301.81], [9E9, 9E9, 9E9, 9E9, 9E9, 9E9]];
	VAR jointtarget CDP_843 := [[12.04, 35.78, 6.23, 0, 47.99, -301.84], [9E9, 9E9, 9E9, 9E9, 9E9, 9E9]];
	VAR jointtarget CDP_844 := [[12.01, 35.8, 6.2, 0, 48, -301.87], [9E9, 9E9, 9E9, 9E9, 9E9, 9E9]];
	VAR jointtarget CDP_845 := [[11.98, 35.82, 6.17, 0, 48.01, -301.89], [9E9, 9E9, 9E9, 9E9, 9E9, 9E9]];
	VAR jointtarget CDP_846 := [[11.95, 35.84, 6.14, 0, 48.03, -301.92], [9E9, 9E9, 9E9, 9E9, 9E9, 9E9]];
	VAR jointtarget CDP_847 := [[11.92, 35.85, 6.1, 0, 48.04, -301.95], [9E9, 9E9, 9E9, 9E9, 9E9, 9E9]];
	VAR jointtarget CDP_848 := [[11.9, 35.87, 6.07, 0, 48.06, -301.98], [9E9, 9E9, 9E9, 9E9, 9E9, 9E9]];
	VAR jointtarget CDP_849 := [[11.87, 35.89, 6.04, 0, 48.07, -302.01], [9E9, 9E9, 9E9, 9E9, 9E9, 9E9]];
	VAR jointtarget CDP_850 := [[11.84, 35.91, 6, 0, 48.08, -302.04], [9E9, 9E9, 9E9, 9E9, 9E9, 9E9]];
	VAR jointtarget CDP_851 := [[11.81, 35.93, 5.97, 0, 48.1, -302.07], [9E9, 9E9, 9E9, 9E9, 9E9, 9E9]];
	VAR jointtarget CDP_852 := [[11.78, 35.95, 5.94, 0, 48.11, -302.09], [9E9, 9E9, 9E9, 9E9, 9E9, 9E9]];
	VAR jointtarget CDP_853 := [[11.75, 35.97, 5.9, 0, 48.12, -302.12], [9E9, 9E9, 9E9, 9E9, 9E9, 9E9]];
	VAR jointtarget CDP_854 := [[11.73, 35.99, 5.87, 0, 48.14, -302.15], [9E9, 9E9, 9E9, 9E9, 9E9, 9E9]];
	VAR jointtarget CDP_855 := [[11.7, 36.01, 5.84, 0, 48.15, -302.18], [9E9, 9E9, 9E9, 9E9, 9E9, 9E9]];
	VAR jointtarget CDP_856 := [[11.67, 36.03, 5.81, 0, 48.17, -302.21], [9E9, 9E9, 9E9, 9E9, 9E9, 9E9]];
	VAR jointtarget CDP_857 := [[11.64, 36.05, 5.77, 0, 48.18, -302.24], [9E9, 9E9, 9E9, 9E9, 9E9, 9E9]];
	VAR jointtarget CDP_858 := [[11.61, 36.07, 5.74, 0, 48.19, -302.27], [9E9, 9E9, 9E9, 9E9, 9E9, 9E9]];
	VAR jointtarget CDP_859 := [[11.58, 36.09, 5.71, 0, 48.21, -302.29], [9E9, 9E9, 9E9, 9E9, 9E9, 9E9]];
	VAR jointtarget CDP_860 := [[11.54, 36.12, 5.65, 0, 48.23, -301.24], [9E9, 9E9, 9E9, 9E9, 9E9, 9E9]];
	VAR jointtarget CDP_861 := [[11.49, 36.15, 5.6, 0, 48.25, -299.1], [9E9, 9E9, 9E9, 9E9, 9E9, 9E9]];
	VAR jointtarget CDP_862 := [[11.44, 36.17, 5.55, 0, 48.27, -296.95], [9E9, 9E9, 9E9, 9E9, 9E9, 9E9]];
	VAR jointtarget CDP_863 := [[11.39, 36.2, 5.51, 0, 48.29, -294.81], [9E9, 9E9, 9E9, 9E9, 9E9, 9E9]];
	VAR jointtarget CDP_864 := [[11.34, 36.22, 5.47, 0, 48.31, -292.67], [9E9, 9E9, 9E9, 9E9, 9E9, 9E9]];
	VAR jointtarget CDP_865 := [[11.28, 36.24, 5.43, 0, 48.32, -290.53], [9E9, 9E9, 9E9, 9E9, 9E9, 9E9]];
	VAR jointtarget CDP_866 := [[11.23, 36.26, 5.4, 0, 48.33, -288.38], [9E9, 9E9, 9E9, 9E9, 9E9, 9E9]];
	VAR jointtarget CDP_867 := [[11.18, 36.28, 5.37, 0, 48.35, -286.24], [9E9, 9E9, 9E9, 9E9, 9E9, 9E9]];
	VAR jointtarget CDP_868 := [[11.13, 36.3, 5.35, 0, 48.36, -284.1], [9E9, 9E9, 9E9, 9E9, 9E9, 9E9]];
	VAR jointtarget CDP_869 := [[11.07, 36.31, 5.33, 0, 48.37, -281.96], [9E9, 9E9, 9E9, 9E9, 9E9, 9E9]];
	VAR jointtarget CDP_870 := [[11.02, 36.32, 5.31, 0, 48.37, -279.82], [9E9, 9E9, 9E9, 9E9, 9E9, 9E9]];
	VAR jointtarget CDP_871 := [[10.96, 36.33, 5.3, 0, 48.38, -277.69], [9E9, 9E9, 9E9, 9E9, 9E9, 9E9]];
	VAR jointtarget CDP_872 := [[10.91, 36.33, 5.29, 0, 48.38, -275.55], [9E9, 9E9, 9E9, 9E9, 9E9, 9E9]];
	VAR jointtarget CDP_873 := [[10.85, 36.34, 5.28, 0, 48.39, -273.41], [9E9, 9E9, 9E9, 9E9, 9E9, 9E9]];
	VAR jointtarget CDP_874 := [[10.8, 36.34, 5.28, 0, 48.39, -271.27], [9E9, 9E9, 9E9, 9E9, 9E9, 9E9]];
	VAR jointtarget CDP_875 := [[10.74, 36.34, 5.28, 0, 48.39, -269.13], [9E9, 9E9, 9E9, 9E9, 9E9, 9E9]];
	VAR jointtarget CDP_876 := [[10.69, 36.33, 5.28, 0, 48.38, -266.99], [9E9, 9E9, 9E9, 9E9, 9E9, 9E9]];
	VAR jointtarget CDP_877 := [[10.63, 36.33, 5.29, 0, 48.38, -264.85], [9E9, 9E9, 9E9, 9E9, 9E9, 9E9]];
	VAR jointtarget CDP_878 := [[10.58, 36.32, 5.31, 0, 48.37, -262.71], [9E9, 9E9, 9E9, 9E9, 9E9, 9E9]];
	VAR jointtarget CDP_879 := [[10.52, 36.31, 5.32, 0, 48.37, -260.58], [9E9, 9E9, 9E9, 9E9, 9E9, 9E9]];
	VAR jointtarget CDP_880 := [[9.44, 36.1, 5.68, 0, 48.22, -260.56], [9E9, 9E9, 9E9, 9E9, 9E9, 9E9]];
	VAR jointtarget CDP_881 := [[8.36, 35.92, 5.99, 0, 48.09, -261.64], [9E9, 9E9, 9E9, 9E9, 9E9, 9E9]];
	VAR jointtarget CDP_882 := [[7.27, 35.76, 6.27, 0, 47.97, -262.73], [9E9, 9E9, 9E9, 9E9, 9E9, 9E9]];
	VAR jointtarget CDP_883 := [[6.17, 35.62, 6.51, 0, 47.87, -263.83], [9E9, 9E9, 9E9, 9E9, 9E9, 9E9]];
	VAR jointtarget CDP_884 := [[5.07, 35.5, 6.71, 0, 47.79, -264.93], [9E9, 9E9, 9E9, 9E9, 9E9, 9E9]];
	VAR jointtarget CDP_885 := [[3.97, 35.41, 6.87, 0, 47.72, -266.03], [9E9, 9E9, 9E9, 9E9, 9E9, 9E9]];
	VAR jointtarget CDP_886 := [[2.86, 35.34, 6.99, 0, 47.67, -267.14], [9E9, 9E9, 9E9, 9E9, 9E9, 9E9]];
	VAR jointtarget CDP_887 := [[1.75, 35.29, 7.07, 0, 47.64, -268.25], [9E9, 9E9, 9E9, 9E9, 9E9, 9E9]];
	VAR jointtarget CDP_888 := [[0.64, 35.27, 7.11, 0, 47.62, -269.36], [9E9, 9E9, 9E9, 9E9, 9E9, 9E9]];
	VAR jointtarget CDP_889 := [[-0.47, 35.26, 7.11, 0, 47.62, -270.47], [9E9, 9E9, 9E9, 9E9, 9E9, 9E9]];
	VAR jointtarget CDP_890 := [[-1.58, 35.29, 7.08, 0, 47.64, -271.58], [9E9, 9E9, 9E9, 9E9, 9E9, 9E9]];
	VAR jointtarget CDP_891 := [[-2.69, 35.33, 7, 0, 47.67, -272.69], [9E9, 9E9, 9E9, 9E9, 9E9, 9E9]];
	VAR jointtarget CDP_892 := [[-3.8, 35.4, 6.89, 0, 47.72, -273.8], [9E9, 9E9, 9E9, 9E9, 9E9, 9E9]];
	VAR jointtarget CDP_893 := [[-4.9, 35.49, 6.73, 0, 47.78, -274.9], [9E9, 9E9, 9E9, 9E9, 9E9, 9E9]];
	VAR jointtarget CDP_894 := [[-6, 35.6, 6.54, 0, 47.86, -276], [9E9, 9E9, 9E9, 9E9, 9E9, 9E9]];
	VAR jointtarget CDP_895 := [[-7.1, 35.73, 6.31, 0, 47.96, -277.1], [9E9, 9E9, 9E9, 9E9, 9E9, 9E9]];
	VAR jointtarget CDP_896 := [[-8.19, 35.89, 6.04, 0, 48.07, -278.19], [9E9, 9E9, 9E9, 9E9, 9E9, 9E9]];
	VAR jointtarget CDP_897 := [[-9.28, 36.07, 5.73, 0, 48.2, -279.28], [9E9, 9E9, 9E9, 9E9, 9E9, 9E9]];
	VAR jointtarget CDP_898 := [[-10.36, 36.28, 5.38, 0, 48.34, -280.36], [9E9, 9E9, 9E9, 9E9, 9E9, 9E9]];
	VAR jointtarget CDP_899 := [[-11.43, 36.5, 4.99, 0, 48.51, -281.43], [9E9, 9E9, 9E9, 9E9, 9E9, 9E9]];
	VAR jointtarget CDP_900 := [[-11.44, 36.51, 4.99, 0, 48.51, -281.78], [9E9, 9E9, 9E9, 9E9, 9E9, 9E9]];
	VAR jointtarget CDP_901 := [[-11.46, 36.51, 4.98, 0, 48.51, -282.45], [9E9, 9E9, 9E9, 9E9, 9E9, 9E9]];
	VAR jointtarget CDP_902 := [[-11.48, 36.51, 4.97, 0, 48.51, -283.13], [9E9, 9E9, 9E9, 9E9, 9E9, 9E9]];
	VAR jointtarget CDP_903 := [[-11.49, 36.52, 4.96, 0, 48.52, -283.81], [9E9, 9E9, 9E9, 9E9, 9E9, 9E9]];
	VAR jointtarget CDP_904 := [[-11.51, 36.52, 4.96, 0, 48.52, -284.49], [9E9, 9E9, 9E9, 9E9, 9E9, 9E9]];
	VAR jointtarget CDP_905 := [[-11.53, 36.53, 4.95, 0, 48.52, -285.17], [9E9, 9E9, 9E9, 9E9, 9E9, 9E9]];
	VAR jointtarget CDP_906 := [[-11.54, 36.53, 4.94, 0, 48.53, -285.84], [9E9, 9E9, 9E9, 9E9, 9E9, 9E9]];
	VAR jointtarget CDP_907 := [[-11.56, 36.54, 4.93, 0, 48.53, -286.52], [9E9, 9E9, 9E9, 9E9, 9E9, 9E9]];
	VAR jointtarget CDP_908 := [[-11.57, 36.54, 4.92, 0, 48.54, -287.2], [9E9, 9E9, 9E9, 9E9, 9E9, 9E9]];
	VAR jointtarget CDP_909 := [[-11.59, 36.55, 4.91, 0, 48.54, -287.88], [9E9, 9E9, 9E9, 9E9, 9E9, 9E9]];
	VAR jointtarget CDP_910 := [[-11.6, 36.55, 4.9, 0, 48.54, -288.56], [9E9, 9E9, 9E9, 9E9, 9E9, 9E9]];
	VAR jointtarget CDP_911 := [[-11.62, 36.56, 4.89, 0, 48.55, -289.23], [9E9, 9E9, 9E9, 9E9, 9E9, 9E9]];
	VAR jointtarget CDP_912 := [[-11.64, 36.57, 4.88, 0, 48.55, -289.91], [9E9, 9E9, 9E9, 9E9, 9E9, 9E9]];
	VAR jointtarget CDP_913 := [[-11.65, 36.57, 4.87, 0, 48.56, -290.59], [9E9, 9E9, 9E9, 9E9, 9E9, 9E9]];
	VAR jointtarget CDP_914 := [[-11.67, 36.58, 4.86, 0, 48.56, -291.27], [9E9, 9E9, 9E9, 9E9, 9E9, 9E9]];
	VAR jointtarget CDP_915 := [[-11.68, 36.59, 4.85, 0, 48.57, -291.94], [9E9, 9E9, 9E9, 9E9, 9E9, 9E9]];
	VAR jointtarget CDP_916 := [[-11.7, 36.59, 4.84, 0, 48.57, -292.62], [9E9, 9E9, 9E9, 9E9, 9E9, 9E9]];
	VAR jointtarget CDP_917 := [[-11.71, 36.6, 4.82, 0, 48.58, -293.3], [9E9, 9E9, 9E9, 9E9, 9E9, 9E9]];
	VAR jointtarget CDP_918 := [[-11.73, 36.61, 4.81, 0, 48.58, -293.98], [9E9, 9E9, 9E9, 9E9, 9E9, 9E9]];
	VAR jointtarget CDP_919 := [[-11.74, 36.62, 4.8, 0, 48.59, -294.65], [9E9, 9E9, 9E9, 9E9, 9E9, 9E9]];
	VAR jointtarget CDP_920 := [[-11.8, 36.65, 4.74, 0, 48.61, -295.04], [9E9, 9E9, 9E9, 9E9, 9E9, 9E9]];
	VAR jointtarget CDP_921 := [[-11.86, 36.68, 4.69, 0, 48.63, -295.11], [9E9, 9E9, 9E9, 9E9, 9E9, 9E9]];
	VAR jointtarget CDP_922 := [[-11.93, 36.71, 4.64, 0, 48.66, -295.17], [9E9, 9E9, 9E9, 9E9, 9E9, 9E9]];
	VAR jointtarget CDP_923 := [[-11.99, 36.74, 4.58, 0, 48.68, -295.23], [9E9, 9E9, 9E9, 9E9, 9E9, 9E9]];
	VAR jointtarget CDP_924 := [[-12.05, 36.77, 4.53, 0, 48.7, -295.29], [9E9, 9E9, 9E9, 9E9, 9E9, 9E9]];
	VAR jointtarget CDP_925 := [[-12.11, 36.8, 4.47, 0, 48.72, -295.35], [9E9, 9E9, 9E9, 9E9, 9E9, 9E9]];
	VAR jointtarget CDP_926 := [[-12.17, 36.84, 4.42, 0, 48.75, -295.41], [9E9, 9E9, 9E9, 9E9, 9E9, 9E9]];
	VAR jointtarget CDP_927 := [[-12.23, 36.87, 4.36, 0, 48.77, -295.47], [9E9, 9E9, 9E9, 9E9, 9E9, 9E9]];
	VAR jointtarget CDP_928 := [[-12.29, 36.9, 4.31, 0, 48.79, -295.53], [9E9, 9E9, 9E9, 9E9, 9E9, 9E9]];
	VAR jointtarget CDP_929 := [[-12.35, 36.93, 4.25, 0, 48.82, -295.59], [9E9, 9E9, 9E9, 9E9, 9E9, 9E9]];
	VAR jointtarget CDP_930 := [[-12.41, 36.96, 4.2, 0, 48.84, -295.65], [9E9, 9E9, 9E9, 9E9, 9E9, 9E9]];
	VAR jointtarget CDP_931 := [[-12.47, 36.99, 4.14, 0, 48.86, -295.71], [9E9, 9E9, 9E9, 9E9, 9E9, 9E9]];
	VAR jointtarget CDP_932 := [[-12.53, 37.03, 4.09, 0, 48.88, -295.77], [9E9, 9E9, 9E9, 9E9, 9E9, 9E9]];
	VAR jointtarget CDP_933 := [[-12.59, 37.06, 4.03, 0, 48.91, -295.83], [9E9, 9E9, 9E9, 9E9, 9E9, 9E9]];
	VAR jointtarget CDP_934 := [[-12.65, 37.09, 3.98, 0, 48.93, -295.89], [9E9, 9E9, 9E9, 9E9, 9E9, 9E9]];
	VAR jointtarget CDP_935 := [[-12.71, 37.12, 3.92, 0, 48.95, -295.95], [9E9, 9E9, 9E9, 9E9, 9E9, 9E9]];
	VAR jointtarget CDP_936 := [[-12.77, 37.16, 3.87, 0, 48.98, -296.01], [9E9, 9E9, 9E9, 9E9, 9E9, 9E9]];
	VAR jointtarget CDP_937 := [[-12.83, 37.19, 3.81, 0, 49, -296.07], [9E9, 9E9, 9E9, 9E9, 9E9, 9E9]];
	VAR jointtarget CDP_938 := [[-12.89, 37.22, 3.75, 0, 49.03, -296.13], [9E9, 9E9, 9E9, 9E9, 9E9, 9E9]];
	VAR jointtarget CDP_939 := [[-12.95, 37.25, 3.7, 0, 49.05, -296.19], [9E9, 9E9, 9E9, 9E9, 9E9, 9E9]];
	VAR jointtarget CDP_940 := [[-13.07, 37.31, 3.61, 0, 49.09, -291.14], [9E9, 9E9, 9E9, 9E9, 9E9, 9E9]];
	VAR jointtarget CDP_941 := [[-13.19, 37.33, 3.56, 0, 49.11, -280.95], [9E9, 9E9, 9E9, 9E9, 9E9, 9E9]];
	VAR jointtarget CDP_942 := [[-13.32, 37.33, 3.56, 0, 49.11, -270.75], [9E9, 9E9, 9E9, 9E9, 9E9, 9E9]];
	VAR jointtarget CDP_943 := [[-13.45, 37.31, 3.6, 0, 49.09, -260.55], [9E9, 9E9, 9E9, 9E9, 9E9, 9E9]];
	VAR jointtarget CDP_944 := [[-13.57, 37.26, 3.68, 0, 49.06, -250.35], [9E9, 9E9, 9E9, 9E9, 9E9, 9E9]];
	VAR jointtarget CDP_945 := [[-13.68, 37.19, 3.81, 0, 49, -240.14], [9E9, 9E9, 9E9, 9E9, 9E9, 9E9]];
	VAR jointtarget CDP_946 := [[-13.78, 37.1, 3.97, 0, 48.94, -229.91], [9E9, 9E9, 9E9, 9E9, 9E9, 9E9]];
	VAR jointtarget CDP_947 := [[-13.86, 36.99, 4.16, 0, 48.86, -219.67], [9E9, 9E9, 9E9, 9E9, 9E9, 9E9]];
	VAR jointtarget CDP_948 := [[-13.93, 36.86, 4.37, 0, 48.77, -209.41], [9E9, 9E9, 9E9, 9E9, 9E9, 9E9]];
	VAR jointtarget CDP_949 := [[-13.97, 36.73, 4.61, 0, 48.67, -199.13], [9E9, 9E9, 9E9, 9E9, 9E9, 9E9]];
	VAR jointtarget CDP_950 := [[-13.99, 36.58, 4.85, 0, 48.57, -188.83], [9E9, 9E9, 9E9, 9E9, 9E9, 9E9]];
	VAR jointtarget CDP_951 := [[-13.98, 36.44, 5.1, 0, 48.46, -178.5], [9E9, 9E9, 9E9, 9E9, 9E9, 9E9]];
	VAR jointtarget CDP_952 := [[-13.96, 36.3, 5.34, 0, 48.36, -168.15], [9E9, 9E9, 9E9, 9E9, 9E9, 9E9]];
	VAR jointtarget CDP_953 := [[-13.91, 36.17, 5.56, 0, 48.27, -157.77], [9E9, 9E9, 9E9, 9E9, 9E9, 9E9]];
	VAR jointtarget CDP_954 := [[-13.84, 36.05, 5.77, 0, 48.18, -147.38], [9E9, 9E9, 9E9, 9E9, 9E9, 9E9]];
	VAR jointtarget CDP_955 := [[-13.75, 35.95, 5.95, 0, 48.11, -136.97], [9E9, 9E9, 9E9, 9E9, 9E9, 9E9]];
	VAR jointtarget CDP_956 := [[-13.64, 35.86, 6.09, 0, 48.05, -126.54], [9E9, 9E9, 9E9, 9E9, 9E9, 9E9]];
	VAR jointtarget CDP_957 := [[-13.52, 35.8, 6.2, 0, 48, -116.09], [9E9, 9E9, 9E9, 9E9, 9E9, 9E9]];
	VAR jointtarget CDP_958 := [[-13.4, 35.76, 6.27, 0, 47.97, -105.64], [9E9, 9E9, 9E9, 9E9, 9E9, 9E9]];
	VAR jointtarget CDP_959 := [[-13.27, 35.75, 6.29, 0, 47.96, -95.19], [9E9, 9E9, 9E9, 9E9, 9E9, 9E9]];
	VAR jointtarget CDP_960 := [[-13.2, 35.75, 6.29, 0, 47.96, -89.96], [9E9, 9E9, 9E9, 9E9, 9E9, 9E9]];
	VAR jointtarget CDP_961 := [[-13.13, 35.75, 6.29, 0, 47.97, -89.89], [9E9, 9E9, 9E9, 9E9, 9E9, 9E9]];
	VAR jointtarget CDP_962 := [[-13.06, 35.74, 6.29, 0, 47.97, -89.82], [9E9, 9E9, 9E9, 9E9, 9E9, 9E9]];
	VAR jointtarget CDP_963 := [[-12.99, 35.74, 6.29, 0, 47.97, -89.75], [9E9, 9E9, 9E9, 9E9, 9E9, 9E9]];
	VAR jointtarget CDP_964 := [[-12.93, 35.74, 6.29, 0, 47.97, -89.69], [9E9, 9E9, 9E9, 9E9, 9E9, 9E9]];
	VAR jointtarget CDP_965 := [[-12.86, 35.74, 6.29, 0, 47.97, -89.62], [9E9, 9E9, 9E9, 9E9, 9E9, 9E9]];
	VAR jointtarget CDP_966 := [[-12.79, 35.74, 6.29, 0, 47.97, -89.55], [9E9, 9E9, 9E9, 9E9, 9E9, 9E9]];
	VAR jointtarget CDP_967 := [[-12.72, 35.74, 6.28, 0, 47.97, -89.48], [9E9, 9E9, 9E9, 9E9, 9E9, 9E9]];
	VAR jointtarget CDP_968 := [[-12.65, 35.74, 6.28, 0, 47.97, -89.41], [9E9, 9E9, 9E9, 9E9, 9E9, 9E9]];
	VAR jointtarget CDP_969 := [[-12.59, 35.74, 6.28, 0, 47.97, -89.35], [9E9, 9E9, 9E9, 9E9, 9E9, 9E9]];
	VAR jointtarget CDP_970 := [[-12.52, 35.74, 6.28, 0, 47.98, -89.28], [9E9, 9E9, 9E9, 9E9, 9E9, 9E9]];
	VAR jointtarget CDP_971 := [[-12.45, 35.75, 6.28, 0, 47.98, -89.21], [9E9, 9E9, 9E9, 9E9, 9E9, 9E9]];
	VAR jointtarget CDP_972 := [[-12.38, 35.75, 6.28, 0, 47.98, -89.14], [9E9, 9E9, 9E9, 9E9, 9E9, 9E9]];
	VAR jointtarget CDP_973 := [[-12.32, 35.75, 6.27, 0, 47.98, -89.07], [9E9, 9E9, 9E9, 9E9, 9E9, 9E9]];
	VAR jointtarget CDP_974 := [[-12.25, 35.75, 6.27, 0, 47.98, -89.01], [9E9, 9E9, 9E9, 9E9, 9E9, 9E9]];
	VAR jointtarget CDP_975 := [[-12.18, 35.75, 6.27, 0, 47.98, -88.94], [9E9, 9E9, 9E9, 9E9, 9E9, 9E9]];
	VAR jointtarget CDP_976 := [[-12.11, 35.75, 6.27, 0, 47.98, -88.87], [9E9, 9E9, 9E9, 9E9, 9E9, 9E9]];
	VAR jointtarget CDP_977 := [[-12.04, 35.75, 6.26, 0, 47.99, -88.8], [9E9, 9E9, 9E9, 9E9, 9E9, 9E9]];
	VAR jointtarget CDP_978 := [[-11.98, 35.75, 6.26, 0, 47.99, -88.74], [9E9, 9E9, 9E9, 9E9, 9E9, 9E9]];
